FOR i:=1 TO 5 DO
	m_spring2Param[i]:=g_spring2Param[i];
	m_spring3Param[i]:=g_spring3Param[i];
	m_spring5Param[i]:=g_spring5Param[i];
END_FOR
m_spring3Param[6]:=g_spring3Param[6];
END_METHOD

METHOD PUBLIC run : BOOL
VAR_IN_OUT CONSTANT
	// active joint position
	i_jntPos :vec7d;
END_VAR
VAR_IN_OUT
	r_gravity :Vec7d;
END_VAR
VAR

	// position of all the active joint
	m_leftJntPos:ARRAY[1..7] OF LREAL;
	m_rightJntPos:ARRAY[1..7] OF LREAL;
	
	// gravity regression matrix
	regMat:ARRAY[1..5,1..16] OF LREAL;
	
	i,j:INT;
END_VAR
getRegMat(m_armIdx,i_jntPos,regMat);

FOR i:=2 TO 6 DO
	r_gravity[i]:=0;
	FOR j:=1 TO 16 DO
		r_gravity[i]:=r_gravity[i]+regMat[i-1,j]*m_gravityParam[j];
	END_FOR
END_FOR
END_METHOD

(*spring force F = preF+k(L-L0)
% torque trq=F*t=preF*t+k*t*(L-L0)=[t, t*(L-L0)]*[preF,k]'
% this function return [t, t(L-L0)]*)
METHOD PROTECTED spring2RegMat : BOOL
VAR_INPUT
	i_q2:LREAL;
END_VAR

VAR
	// spring paramters
	L0, b1, b2, l1, r0 : LREAL;

	theta,length,t:LREAL;  
	
END_VAR

VAR_OUTPUT
	o_preF:LREAL;
	o_stiff:LREAL;
END_VAR
L0:=m_spring2Param[1]; 
b1:=m_spring2Param[2]; 
b2:=m_spring2Param[3]; 
l1:=m_spring2Param[4]; 
r0:=m_spring2Param[5]; 

L0:=L0+b1+b2;
 
//spring length
theta:=i_q2+90*g_deg2Rad;
length:=SQRT(l1*l1+r0*r0+2*l1*r0*COS(theta));

//force arm
t:=r0*l1*SIN(theta)/Length;

//torque direction is determined by theta(or t)
o_preF:=t;
o_stiff:=t*(length-L0);
END_METHOD

(*spring force F = preF+k(L-L0)
% torque trq=F*t=preF*t+k*t*(L-L0)=[t, t*(L-L0)]*[preF,k]'
% this function return [t, t(L-L0)]*)
METHOD PROTECTED spring3RegMat : BOOL
VAR_INPUT
	i_q3:LREAL;
END_VAR

VAR
	// spring paramters
	L0, b1, b2, l1, r0, d: LREAL;

	alpha, beta,tanBeta, length,t:LREAL;  
	
	spring: INT;
END_VAR

VAR_OUTPUT
	o_preF:LREAL;
	o_stiff:LREAL;
END_VAR
L0:=m_spring3Param[1]; 
b1:=m_spring3Param[2]; 
b2:=m_spring3Param[3]; 
l1:=m_spring3Param[4]; 
r0:=m_spring3Param[5];
d:=m_spring3Param[6];

L0:=L0+b1+b2;
 
// spring length
    alpha:=i_q3+90*g_deg2Rad;
    tanBeta:=(r0*SIN(alpha)+d)/(l1+r0*COS(alpha));
    beta:=ATAN(tanBeta);
    length:=d/SIN(beta)+r0*SIN(alpha)/SIN(beta);
    
// force arm
    t:=(l1-d*cot(beta))*SIN(beta);
    
// torque direction is determined by theta(or t)
    o_preF:=t;
    o_stiff:=t*(length-L0);
END_METHOD

(*spring force F = preF+k(L-L0)
 torque trq=F*t=preF*t+k*t*(L-L0)=[t, t*(L-L0)]*[preF,k]'
 this function return [t, t(L-L0)]
 armIdx, 0 for left arm , 1 for right arm]*)
METHOD PROTECTED spring5RegMat : BOOL
VAR_INPUT
	i_q5:LREAL;
END_VAR

VAR
	// spring paramters
	L0, s1, L1, r0, beta: LREAL;

	theta, length,t:LREAL;  
	
	spring: INT;
	joint: INT;
	armIdx: INT;
	b1: LREAL;
END_VAR

VAR_OUTPUT
	o_preF:LREAL;
	o_stiff:LREAL;
END_VAR
L0:=m_spring5Param[1]; 
s1:=m_spring5Param[2]; 
L1:=m_spring5Param[3]; 
r0:=m_spring5Param[4]; 
beta:=m_spring5Param[5];

L0:=L0+s1;
 
// joint 5 motion angle
IF 1=m_armIdx THEN 
	theta:=i_q5-pi;// left arm
ELSE
	theta:=pi-i_q5; // right arm
END_IF

// spring length and force arm
length:=SQRT(L1*L1+r0*r0+2*L1*r0*COS(theta+beta));
t:=L1*r0*SIN(theta+beta)/length;

// torque direction is determined by t
IF 1=m_armIdx THEN 
	o_preF:=t;
	o_stiff:=t*(length-L0);
else
	o_preF:=-t;
	o_stiff:=-t*(length-L0);
END_IF
END_METHOD

END_FUNCTION_BLOCK

// ---- FBs_RobotDynamics/FB_MasterDynamic.TcPOU
FUNCTION_BLOCK FB_MasterDynamic
VAR_INPUT
END_VAR
VAR_OUTPUT
END_VAR
VAR
	m_armIdx :INT;
	//kinematic constraint
	//  q3 = q8 - q2;            qdot3=qdot8-qdot2;
	//  q9 = q2-q8;              qdot9=qdot2-qdot8;
	//  q4= q4motor+q8-q2-90;    qdot4=qdot4m+qdot8
 	// jacobian with active joints
 	// jaco_DH*qdot_DH = jaco_DH * (A * qdot_active)= jaco * qdot_active
 	// q_DH=[q1,q2,q3,q4,q5,q6,q7,q8,q9];
 	// q_active=[q1,q2,q8,q4m,q5,q6,q7]
	m_jacoA :ARRAY[1..9,1..7] OF LREAL:=
		[   1,  0,  0,  0,  0,  0,  0,
			0,  1,  0,  0,  0,  0,  0,
			0, -1,  1,  0,  0,  0,  0,
			0, -1,  1,  1,  0,  0,  0,
			0,  0,  0,  0,  1,  0,  0,
			0,  0,  0,  0,  0,  1,  0,
			0,  0,  0,  0,  0,  0,  1,
			0,  0,  1,  0,  0,  0,  0,
			0,  1, -1,  0,  0,  0,  0];
	
	// DH parameters
	m_armDH:ARRAY[1..9] OF Vec4d;// last column is joint position
	m_d1, m_a3,m_a4,m_d4,m_a9 :LREAL;
	
	// dynamic parameters
	m_linkMass :ARRAY[1..9] OF LREAL;
	m_linkCOM :ARRAY[1..9] OF Vec3d;
	m_linkInertia :ARRAY[1..9] OF Mat3d;
		
	// frame of each joint
	m_jntFrame :ARRAY[1..9] OF ST_Frame;
	
	// jacobian of mass center
	m_Jp :ARRAY[1..9] OF Mat37;
	m_Jo :ARRAY[1..9] OF Mat37;
	
	// tcp jacobian
	m_jaco : Mat67;
	
	// motor inertia at link size
	m_motorInertia :Vec7d;
	
	// mass matrix in joint space
	m_massMat :Mat7d;
	m_massMatInv:Mat7d;
	
	// mass matrix in cartesian space
	m_lambdaInv :Mat6d;
	m_lambda :Mat6d;
	
	// dynamic nullspace(I-J'*inv(J'))
	m_JtGeneInv :Mat67;
	m_dynaNullspace : Mat7d;
	
END_VAR

PROPERTY PUBLIC cartMassMat : Mat6d
GET
cartMassMat := m_lambda;
END_GET
END_PROPERTY

PROPERTY PUBLIC dynaNullspace : Mat7d
GET
dynaNullspace:=m_dynaNullspace;
END_GET
END_PROPERTY

METHOD init : BOOL
VAR_INPUT
	i_armIdx :INT ;
END_VAR

VAR
	i:INT;
END_VAR
m_armIdx:=i_armIdx;
m_d1:=g_d1;
m_a3:=g_a3;
m_a4:=g_a4;
m_d4:=g_d4;
m_a9:=g_a9;

m_linkMass:=g_linkMass;
FOR i:=1 TO 9 DO
	m_linkCOM[i][1]:=g_linkCOM[i,1];
	m_linkCOM[i][2]:=g_linkCOM[i,2];
	m_linkCOM[i][3]:=g_linkCOM[i,3];
	
	m_armDH[i][1]:=g_masterArmDH[i,1];
	m_armDH[i][2]:=g_masterArmDH[i,2];
	m_armDH[i][3]:=g_masterArmDH[i,3];
	m_armDH[i][4]:=g_masterArmDH[i,4];
	
	m_linkInertia[i][1,1]:=g_linkInertia[i,1];
	m_linkInertia[i][2,2]:=g_linkInertia[i,2];
	m_linkInertia[i][3,3]:=g_linkInertia[i,3];
	m_linkInertia[i][1,2]:=g_linkInertia[i,4];
	m_linkInertia[i][1,3]:=g_linkInertia[i,5];
	m_linkInertia[i][2,3]:=g_linkInertia[i,6];
	m_linkInertia[i][2,1]:=m_linkInertia[i][1,2];
	m_linkInertia[i][3,1]:=m_linkInertia[i][1,3];
	m_linkInertia[i][3,2]:=m_linkInertia[i][2,3];
END_FOR

FOR i:=1 TO 7 DO
	m_motorInertia[i]:=g_motorInertia[i]*g_motorReduction[i]*g_motorReduction[i];
END_FOR
END_METHOD

PROPERTY PUBLIC jntMassMat : Mat7d
GET
jntMassMat := m_massMat;
END_GET
END_PROPERTY

// update dynamic and kinematic data 
METHOD updateDynamic : BOOL
VAR_IN_OUT CONSTANT
	i_jntPos : Vec7d;
END_VAR
VAR
	
	i,j:INT;
	m,n :INT;
	linkMassMat :ARRAY[1..9] OF Mat7d;
	linkInerMat :ARRAY[1..9] OF Mat7d;
	inertia,Rt :Mat3d;
	JotI :ARRAY[1..7,1..3] OF LREAL;
	Jot :ARRAY[1..7,1..3] OF LREAL;
	Jpt :ARRAY[1..7,1..3] OF LREAL;
	
	tmpMat3d :Mat3d;
	tmpMat67: Mat67;
	tmpMat7d : Mat7d;
	jacoT: Mat76;
	
END_VAR
// update kinematic 
updateKinematic(i_jntPos);

// joint space mass matrix
// massMat=m*Jp'*Jp+Jo'*R*I*R'*Jo
FOR i:=1 TO 9 DO
	// iner=R*I*R'
	matMultiply(m_jntFrame[i].m_rot,m_linkInertia[i],tmpMat3d);
	matTranspose(m_jntFrame[i].m_rot, Rt);
	matMultiply(tmpMat3d,Rt,inertia);
	
	// m*Jp'*Jp+Jo'*iner*Jo
	matTranspose(m_Jp[i],Jpt);
	matMultiply(Jpt,m_Jp[i], tmpMat7d);
	matMultiNum(tmpMat7d, m_linkMass[i],linkMassMat[i]);
	
	matTranspose(m_Jo[i],Jot);
	matMultiply(Jot,inertia, JotI);
	matMultiply(JotI,m_Jo[i],linkInerMat[i]);
END_FOR

// total mass mat
m_massMat :=g_zeroMat7d;
FOR i:=1 TO 9 DO
	matSelfAdd(m_massMat,linkMassMat[i]);
	matSelfAdd(m_massMat,linkInerMat[i]);
END_FOR

// add motor inertial 
FOR i:=1 TO 7 DO
	m_massMat[i,i]:=m_massMat[i,i]+m_motorInertia[i];
END_FOR

// mass mat inverse
invMat7(m_massMat,m_massMatInv);

// cartesian mass matrix
matTranspose(m_jaco, jacoT);
matMultiply(m_jaco,m_massMatInv, tmpMat67);
matMultiply(tmpMat67, jacoT, m_lambdaInv);
invMat6(m_lambdaInv, m_lambda);

// dyanmic nullspace
matMultiply(m_lambda, m_jaco, tmpMat67);
matMultiply(tmpMat67, m_massMatInv, m_JtGeneInv);
matMultiply(jacoT,m_JtGeneInv,tmpMat7d);
matSub(g_eye7d, tmpMat7d, m_dynaNullspace);
END_METHOD

// only update kinematic data
METHOD PUBLIC updateKinematic : BOOL
VAR_IN_OUT CONSTANT
	i_jntPos : Vec7d;
END_VAR
VAR
	Jp :ARRAY[1..3, 1..9] OF LREAL:=[27(0)];
	Jo :ARRAY[1..3, 1..9] OF LREAL:=[27(0)];
	jacoDH :Mat67;
	T :ST_Frame;
	i,j:INT;
	Pc,z,p:Vec3d;
	tcpPos :Vec3d;
	m,n :INT;
	
END_VAR
// tranform a joint positon to DH ones
m_armDH[1][4]:=i_jntPos[1];
m_armDH[2][4]:=i_jntPos[2];
m_armDH[3][4]:=i_jntPos[3]-i_jntPos[2];
m_armDH[4][4]:=i_jntPos[4]+i_jntPos[3]-i_jntPos[2]-pi/2;
m_armDH[5][4]:=i_jntPos[5];
m_armDH[6][4]:=i_jntPos[6];
m_armDH[7][4]:=i_jntPos[7];
m_armDH[8][4]:=i_jntPos[3];
m_armDH[9][4]:=i_jntPos[2]-i_jntPos[3];

// compute joint frame
m_jntFrame[1]:=DHTrans(m_armDH[1]);
T:=DHTrans(m_armDH[2]);
m_jntFrame[2]:=transform(m_jntFrame[1],T);
T:=DHTrans(m_armDH[3]);
m_jntFrame[3]:=transform(m_jntFrame[2],T);
T:=DHTrans(m_armDH[4]);
m_jntFrame[4]:=transform(m_jntFrame[3],T);
T:=DHTrans(m_armDH[5]);
m_jntFrame[5]:=transform(m_jntFrame[4],T);
T:=DHTrans(m_armDH[6]);
m_jntFrame[6]:=transform(m_jntFrame[5],T);
T:=DHTrans(m_armDH[7]);
m_jntFrame[7]:=transform(m_jntFrame[6],T);
T:=DHTrans(m_armDH[8]);
m_jntFrame[8]:=transform(m_jntFrame[1],T);
T:=DHTrans(m_armDH[9]);
m_jntFrame[9]:=transform(m_jntFrame[8],T);

// tcp jacobian
tcpPos:=m_jntFrame[7].m_pos;
FOR i:=1 TO 7 DO
	T:=m_jntFrame[i];
	z[1]:=T.m_rot[1,3];
	z[2]:=T.m_rot[2,3];
	z[3]:=T.m_rot[3,3];
	p:=subVec3(tcpPos,T.m_pos);
	p:=cross(z,p);
	jacoDH[1,i]:=p[1];
	jacoDH[2,i]:=p[2];
	jacoDH[3,i]:=p[3];
	jacoDH[4,i]:=z[1];
	jacoDH[5,i]:=z[2];
	jacoDH[6,i]:=z[3];
END_FOR
// multiply m_jacoA
FOR m:=1 TO 6 DO 
	FOR n:=1 TO 7 DO
		IF 2=n THEN
			m_Jaco[m,n]:=jacoDH[m,2]-jacoDH[m,3]-jacoDH[m,4];
		ELSIF 3 =n THEN
			m_Jaco[m,n]:=jacoDH[m,3]+jacoDH[m,4];
		ELSE
			m_Jaco[m,n]:=jacoDH[m,n];
		END_IF
	END_FOR
END_FOR


// jacobian of mass center
FOR i:=1 TO 9 DO 
    T:=m_jntFrame[i];
	// mass center world position
    Pc:=mat3Vec3(T.m_rot,m_linkCOM[i]);
	Pc:=addVec3(Pc,T.m_pos);
    FOR j:=1 TO i DO
        IF (i>7 AND j>1 AND j<8) THEN
			Jp[1,j]:=0;
			Jp[2,j]:=0;
			Jp[3,j]:=0;
			Jo[1,j]:=0;
			Jo[2,j]:=0;
			Jo[3,j]:=0;
            CONTINUE;
        END_IF
        T:=m_jntFrame[j];
		z[1]:=T.m_rot[1,3];
		z[2]:=T.m_rot[2,3];
		z[3]:=T.m_rot[3,3];
        p:=subVec3(Pc,T.m_pos);
		p:=cross(z,p);
		Jp[1,j]:=p[1];
		Jp[2,j]:=p[2];
		Jp[3,j]:=p[3];
        Jo[1,j]:=z[1];
		Jo[2,j]:=z[2];
		Jo[3,j]:=z[3];
    END_FOR
	// multiply m_jacoA
	FOR m:=1 TO 3 DO 
		FOR n:=1 TO 7 DO
			IF 2=n THEN
				m_Jp[i][m,n]:=Jp[m,2]-Jp[m,3]-Jp[m,4]+Jp[m,9];
				m_Jo[i][m,n]:=Jo[m,2]-Jo[m,3]-Jo[m,4]+Jo[m,9];
			ELSIF 3 =n THEN
				m_Jp[i][m,n]:=Jp[m,3]+Jp[m,4]+Jp[m,8]-Jp[m,9];
				m_Jo[i][m,n]:=Jo[m,3]+Jo[m,4]+Jo[m,8]-Jo[m,9];
			ELSE
				m_Jp[i][m,n]:=Jp[m,n];
				m_Jo[i][m,n]:=Jo[m,n];
			END_IF
		END_FOR
	END_FOR
END_FOR
END_METHOD

END_FUNCTION_BLOCK

// ---- MatrixLib/matMultiply.TcPOU
// matC = matA * matB
FUNCTION matMultiply : BOOL
VAR_IN_OUT CONSTANT
	matA :ARRAY[*,*] OF LREAL;//m*p
	matB :ARRAY[*,*] OF LREAL;//p*n
END_VAR

VAR_IN_OUT 
	matC :ARRAY[*,*] OF LREAL;//m*n
END_VAR

VAR
	i,j, k :DINT;
	m,n,p :DINT;
	tmp:LREAL;
 
END_VAR

m:=UPPER_BOUND(matA,1);
p:=UPPER_BOUND(matA,2);
n:=UPPER_BOUND(matB,2);

FOR i:=1 TO m DO
	FOR j:=1 TO n DO
		matC[i,j]:=0.0;
	END_FOR
END_FOR

FOR i:=1 TO m DO
	FOR k:=1 TO p DO
		tmp:=matA[i,k];
		FOR j:=1 TO n DO 
		matC[i,j]:=matC[i,j]+tmp*matB[k,j];
		END_FOR
	END_FOR
END_FOR

END_FUNCTION

// ---- MatrixLib/matTranspose.TcPOU
// B =A'
FUNCTION matTranspose : BOOL
VAR_IN_OUT CONSTANT
	matA :ARRAY[*,*] OF LREAL;
END_VAR

VAR_IN_OUT 
	matB :ARRAY[*,*] OF LREAL;
END_VAR

VAR
	i,j:DINT;
	m,n :DINT;
 
END_VAR

m:=UPPER_BOUND(matB,1);
n:= UPPER_BOUND(matB,2);
FOR i:=1 TO m DO
	FOR j:=1 TO n DO
		matB[i,j]:=matA[j,i];
	END_FOR
END_FOR

END_FUNCTION

// ---- MatrixLib/matMultiNum.TcPOU
// matB=num*MatA
FUNCTION matMultiNum : BOOL
VAR_IN_OUT CONSTANT
	matA :ARRAY[*,*] OF LREAL;
	num : LREAL;
END_VAR

VAR_IN_OUT 
	matB :ARRAY[*,*] OF LREAL;
END_VAR

VAR
	m,n :DINT;
	i,j, k :DINT;
 
END_VAR

m:=UPPER_BOUND(matB,1);
n:= UPPER_BOUND(matB,2);
FOR i:=1 TO m DO
	FOR j:=1 TO n DO
		matB[i,j]:=num*matA[i,j];
	END_FOR
END_FOR

END_FUNCTION

// ---- MatrixLib/invMat7.TcPOU
FUNCTION invMat7 : bool
VAR_IN_OUT CONSTANT
	mat :Mat7d;
END_VAR

VAR_IN_OUT
	invMat :Mat7d;
END_VAR
VAR
	dim : INT :=7;
	i,j,k,h:INT;
	m,n :INT;
	cofactorMat : Mat6d;
	adjointMat :Mat7d;
	matDet :LREAL;
END_VAR

matDet :=Det7(mat);
IF matDet=0 THEN
	invMat7:=FALSE;
	RETURN;
END_IF

FOR i :=1 TO dim DO
	FOR j:=1 TO dim DO
		// get cofactor mat
		m:=1;
		n:=1;
		FOR k:=1 TO dim DO
			FOR h:=1 TO dim DO
				IF k<>i AND h <> j THEN
					cofactorMat[m,n]:=mat[k,h];
					n:=n+1;
					IF n>=dim THEN
						m:=m+1;
						n:=1;
					END_IF
				END_IF
			END_FOR
		END_FOR
		
		adjointMat[i,j]:=EXPT(-1,i+j)*Det6(cofactorMat);
	END_FOR
END_FOR

FOR i :=1 TO dim DO
	FOR j:=1 TO dim DO
		invMat[i,j]:=adjointMat[j,i]/matDet;
	END_FOR
END_FOR
invMat7:=true;

END_FUNCTION

// ---- MatrixLib/Det7.TcPOU
FUNCTION Det7 : LREAL
VAR_IN_OUT CONSTANT
	mat: Mat7d;
END_VAR
VAR
	dim : INT :=7;
	i,j,k:INT;
	m,n :INT;
	cofactorMat : Mat6d;
END_VAR

Det7:=0;
FOR i :=1 TO dim DO
	// get cofactor mat
	m:=1;
	n:=1;
	FOR j:=1 TO dim DO
		FOR k:=1 TO dim DO
			IF j<>1 AND k <> i THEN
				cofactorMat[m,n]:=mat[j,k];
				n:=n+1;
				IF n>=dim THEN
					m:=m+1;
					n:=1;
				END_IF
			END_IF
		END_FOR
	END_FOR
	
	Det7:=Det7+ mat[1,i]*EXPT(-1,1+i)*Det6(cofactorMat);
END_FOR

END_FUNCTION

// ---- MatrixLib/Det6.TcPOU
FUNCTION Det6 : LREAL
VAR_IN_OUT CONSTANT
	mat: Mat6d;
END_VAR
VAR
	a11,a12,a13,a14,a15,a16:LREAL;
	a21,a22,a23,a24,a25,a26:LREAL;
	a31,a32,a33,a34,a35,a36:LREAL;
	a41,a42,a43,a44,a45,a46:LREAL;
	a51,a52,a53,a54,a55,a56:LREAL;
	a61,a62,a63,a64,a65,a66:LREAL;
END_VAR


a11:=mat[1,1];
a12:=mat[1,2];
a13:=mat[1,3];
a14:=mat[1,4];
a15:=mat[1,5];
a16:=mat[1,6];

a21:=mat[2,1];
a22:=mat[2,2];
a23:=mat[2,3];
a24:=mat[2,4];
a25:=mat[2,5];
a26:=mat[2,6];

a31:=mat[3,1];
a32:=mat[3,2];
a33:=mat[3,3];
a34:=mat[3,4];
a35:=mat[3,5];
a36:=mat[3,6];

a41:=mat[4,1];
a42:=mat[4,2];
a43:=mat[4,3];
a44:=mat[4,4];
a45:=mat[4,5];
a46:=mat[4,6];

a51:=mat[5,1];
a52:=mat[5,2];
a53:=mat[5,3];
a54:=mat[5,4];
a55:=mat[5,5];
a56:=mat[5,6];

a61:=mat[6,1];
a62:=mat[6,2];
a63:=mat[6,3];
a64:=mat[6,4];
a65:=mat[6,5];
a66:=mat[6,6];

//Det6:=a11*a22*a33*a44*a55*a66 - a11*a22*a33*a44*a56*a65 - a11*a22*a33*a45*a54*a66 + a11*a22*a33*a45*a56*a64 + a11*a22*a33*a46*a54*a65 - a11*a22*a33*a46*a55*a64 - a11*a22*a34*a43*a55*a66 + a11*a22*a34*a43*a56*a65 + a11*a22*a34*a45*a53*a66 - a11*a22*a34*a45*a56*a63 - a11*a22*a34*a46*a53*a65 + a11*a22*a34*a46*a55*a63 + a11*a22*a35*a43*a54*a66 - a11*a22*a35*a43*a56*a64 - a11*a22*a35*a44*a53*a66 + a11*a22*a35*a44*a56*a63 + a11*a22*a35*a46*a53*a64 - a11*a22*a35*a46*a54*a63 - a11*a22*a36*a43*a54*a65 + a11*a22*a36*a43*a55*a64 + a11*a22*a36*a44*a53*a65 - a11*a22*a36*a44*a55*a63 - a11*a22*a36*a45*a53*a64 + a11*a22*a36*a45*a54*a63 - a11*a23*a32*a44*a55*a66 + a11*a23*a32*a44*a56*a65 + a11*a23*a32*a45*a54*a66 - a11*a23*a32*a45*a56*a64 - a11*a23*a32*a46*a54*a65 + a11*a23*a32*a46*a55*a64 + a11*a23*a34*a42*a55*a66 - a11*a23*a34*a42*a56*a65 - a11*a23*a34*a45*a52*a66 + a11*a23*a34*a45*a56*a62 + a11*a23*a34*a46*a52*a65 - a11*a23*a34*a46*a55*a62 - a11*a23*a35*a42*a54*a66 + a11*a23*a35*a42*a56*a64 + a11*a23*a35*a44*a52*a66 - a11*a23*a35*a44*a56*a62 - a11*a23*a35*a46*a52*a64 + a11*a23*a35*a46*a54*a62 + a11*a23*a36*a42*a54*a65 - a11*a23*a36*a42*a55*a64 - a11*a23*a36*a44*a52*a65 + a11*a23*a36*a44*a55*a62 + a11*a23*a36*a45*a52*a64 - a11*a23*a36*a45*a54*a62 + a11*a24*a32*a43*a55*a66 - a11*a24*a32*a43*a56*a65 - a11*a24*a32*a45*a53*a66 + a11*a24*a32*a45*a56*a63 + a11*a24*a32*a46*a53*a65 - a11*a24*a32*a46*a55*a63 - a11*a24*a33*a42*a55*a66 + a11*a24*a33*a42*a56*a65 + a11*a24*a33*a45*a52*a66 - a11*a24*a33*a45*a56*a62 - a11*a24*a33*a46*a52*a65 + a11*a24*a33*a46*a55*a62 + a11*a24*a35*a42*a53*a66 - a11*a24*a35*a42*a56*a63 - a11*a24*a35*a43*a52*a66 + a11*a24*a35*a43*a56*a62 + a11*a24*a35*a46*a52*a63 - a11*a24*a35*a46*a53*a62 - a11*a24*a36*a42*a53*a65 + a11*a24*a36*a42*a55*a63 + a11*a24*a36*a43*a52*a65 - a11*a24*a36*a43*a55*a62 - a11*a24*a36*a45*a52*a63 + a11*a24*a36*a45*a53*a62 - a11*a25*a32*a43*a54*a66 + a11*a25*a32*a43*a56*a64 + a11*a25*a32*a44*a53*a66 - a11*a25*a32*a44*a56*a63 - a11*a25*a32*a46*a53*a64 + a11*a25*a32*a46*a54*a63 + a11*a25*a33*a42*a54*a66 - a11*a25*a33*a42*a56*a64 - a11*a25*a33*a44*a52*a66 + a11*a25*a33*a44*a56*a62 + a11*a25*a33*a46*a52*a64 - a11*a25*a33*a46*a54*a62 - a11*a25*a34*a42*a53*a66 + a11*a25*a34*a42*a56*a63 + a11*a25*a34*a43*a52*a66 - a11*a25*a34*a43*a56*a62 - a11*a25*a34*a46*a52*a63 + a11*a25*a34*a46*a53*a62 + a11*a25*a36*a42*a53*a64 - a11*a25*a36*a42*a54*a63 - a11*a25*a36*a43*a52*a64 + a11*a25*a36*a43*a54*a62 + a11*a25*a36*a44*a52*a63 - a11*a25*a36*a44*a53*a62 + a11*a26*a32*a43*a54*a65 - a11*a26*a32*a43*a55*a64 - a11*a26*a32*a44*a53*a65 + a11*a26*a32*a44*a55*a63 + a11*a26*a32*a45*a53*a64 - a11*a26*a32*a45*a54*a63 - a11*a26*a33*a42*a54*a65 + a11*a26*a33*a42*a55*a64 + a11*a26*a33*a44*a52*a65 - a11*a26*a33*a44*a55*a62 - a11*a26*a33*a45*a52*a64 + a11*a26*a33*a45*a54*a62 + a11*a26*a34*a42*a53*a65 - a11*a26*a34*a42*a55*a63 - a11*a26*a34*a43*a52*a65 + a11*a26*a34*a43*a55*a62 + a11*a26*a34*a45*a52*a63 - a11*a26*a34*a45*a53*a62 - a11*a26*a35*a42*a53*a64 + a11*a26*a35*a42*a54*a63 + a11*a26*a35*a43*a52*a64 - a11*a26*a35*a43*a54*a62 - a11*a26*a35*a44*a52*a63 + a11*a26*a35*a44*a53*a62 - a12*a21*a33*a44*a55*a66 + a12*a21*a33*a44*a56*a65 + a12*a21*a33*a45*a54*a66 - a12*a21*a33*a45*a56*a64 - a12*a21*a33*a46*a54*a65 + a12*a21*a33*a46*a55*a64 + a12*a21*a34*a43*a55*a66 - a12*a21*a34*a43*a56*a65 - a12*a21*a34*a45*a53*a66 + a12*a21*a34*a45*a56*a63 + a12*a21*a34*a46*a53*a65 - a12*a21*a34*a46*a55*a63 - a12*a21*a35*a43*a54*a66 + a12*a21*a35*a43*a56*a64 + a12*a21*a35*a44*a53*a66 - a12*a21*a35*a44*a56*a63 - a12*a21*a35*a46*a53*a64 + a12*a21*a35*a46*a54*a63 + a12*a21*a36*a43*a54*a65 - a12*a21*a36*a43*a55*a64 - a12*a21*a36*a44*a53*a65 + a12*a21*a36*a44*a55*a63 + a12*a21*a36*a45*a53*a64 - a12*a21*a36*a45*a54*a63 + a12*a23*a31*a44*a55*a66 - a12*a23*a31*a44*a56*a65 - a12*a23*a31*a45*a54*a66 + a12*a23*a31*a45*a56*a64 + a12*a23*a31*a46*a54*a65 - a12*a23*a31*a46*a55*a64 - a12*a23*a34*a41*a55*a66 + a12*a23*a34*a41*a56*a65 + a12*a23*a34*a45*a51*a66 - a12*a23*a34*a45*a56*a61 - a12*a23*a34*a46*a51*a65 + a12*a23*a34*a46*a55*a61 + a12*a23*a35*a41*a54*a66 - a12*a23*a35*a41*a56*a64 - a12*a23*a35*a44*a51*a66 + a12*a23*a35*a44*a56*a61 + a12*a23*a35*a46*a51*a64 - a12*a23*a35*a46*a54*a61 - a12*a23*a36*a41*a54*a65 + a12*a23*a36*a41*a55*a64 + a12*a23*a36*a44*a51*a65 - a12*a23*a36*a44*a55*a61 - a12*a23*a36*a45*a51*a64 + a12*a23*a36*a45*a54*a61 - a12*a24*a31*a43*a55*a66 + a12*a24*a31*a43*a56*a65 + a12*a24*a31*a45*a53*a66 - a12*a24*a31*a45*a56*a63 - a12*a24*a31*a46*a53*a65 + a12*a24*a31*a46*a55*a63 + a12*a24*a33*a41*a55*a66 - a12*a24*a33*a41*a56*a65 - a12*a24*a33*a45*a51*a66 + a12*a24*a33*a45*a56*a61 + a12*a24*a33*a46*a51*a65 - a12*a24*a33*a46*a55*a61 - a12*a24*a35*a41*a53*a66 + a12*a24*a35*a41*a56*a63 + a12*a24*a35*a43*a51*a66 - a12*a24*a35*a43*a56*a61 - a12*a24*a35*a46*a51*a63 + a12*a24*a35*a46*a53*a61 + a12*a24*a36*a41*a53*a65 - a12*a24*a36*a41*a55*a63 - a12*a24*a36*a43*a51*a65 + a12*a24*a36*a43*a55*a61 + a12*a24*a36*a45*a51*a63 - a12*a24*a36*a45*a53*a61 + a12*a25*a31*a43*a54*a66 - a12*a25*a31*a43*a56*a64 - a12*a25*a31*a44*a53*a66 + a12*a25*a31*a44*a56*a63 + a12*a25*a31*a46*a53*a64 - a12*a25*a31*a46*a54*a63 - a12*a25*a33*a41*a54*a66 + a12*a25*a33*a41*a56*a64 + a12*a25*a33*a44*a51*a66 - a12*a25*a33*a44*a56*a61 - a12*a25*a33*a46*a51*a64 + a12*a25*a33*a46*a54*a61 + a12*a25*a34*a41*a53*a66 - a12*a25*a34*a41*a56*a63 - a12*a25*a34*a43*a51*a66 + a12*a25*a34*a43*a56*a61 + a12*a25*a34*a46*a51*a63 - a12*a25*a34*a46*a53*a61 - a12*a25*a36*a41*a53*a64 + a12*a25*a36*a41*a54*a63 + a12*a25*a36*a43*a51*a64 - a12*a25*a36*a43*a54*a61 - a12*a25*a36*a44*a51*a63 + a12*a25*a36*a44*a53*a61 - a12*a26*a31*a43*a54*a65 + a12*a26*a31*a43*a55*a64 + a12*a26*a31*a44*a53*a65 - a12*a26*a31*a44*a55*a63 - a12*a26*a31*a45*a53*a64 + a12*a26*a31*a45*a54*a63 + a12*a26*a33*a41*a54*a65 - a12*a26*a33*a41*a55*a64 - a12*a26*a33*a44*a51*a65 + a12*a26*a33*a44*a55*a61 + a12*a26*a33*a45*a51*a64 - a12*a26*a33*a45*a54*a61 - a12*a26*a34*a41*a53*a65 + a12*a26*a34*a41*a55*a63 + a12*a26*a34*a43*a51*a65 - a12*a26*a34*a43*a55*a61 - a12*a26*a34*a45*a51*a63 + a12*a26*a34*a45*a53*a61 + a12*a26*a35*a41*a53*a64 - a12*a26*a35*a41*a54*a63 - a12*a26*a35*a43*a51*a64 + a12*a26*a35*a43*a54*a61 + a12*a26*a35*a44*a51*a63 - a12*a26*a35*a44*a53*a61 + a13*a21*a32*a44*a55*a66 - a13*a21*a32*a44*a56*a65 - a13*a21*a32*a45*a54*a66 + a13*a21*a32*a45*a56*a64 + a13*a21*a32*a46*a54*a65 - a13*a21*a32*a46*a55*a64 - a13*a21*a34*a42*a55*a66 + a13*a21*a34*a42*a56*a65 + a13*a21*a34*a45*a52*a66 - a13*a21*a34*a45*a56*a62 - a13*a21*a34*a46*a52*a65 + a13*a21*a34*a46*a55*a62 + a13*a21*a35*a42*a54*a66 - a13*a21*a35*a42*a56*a64 - a13*a21*a35*a44*a52*a66 + a13*a21*a35*a44*a56*a62 + a13*a21*a35*a46*a52*a64 - a13*a21*a35*a46*a54*a62 - a13*a21*a36*a42*a54*a65 + a13*a21*a36*a42*a55*a64 + a13*a21*a36*a44*a52*a65 - a13*a21*a36*a44*a55*a62 - a13*a21*a36*a45*a52*a64 + a13*a21*a36*a45*a54*a62 - a13*a22*a31*a44*a55*a66 + a13*a22*a31*a44*a56*a65 + a13*a22*a31*a45*a54*a66 - a13*a22*a31*a45*a56*a64 - a13*a22*a31*a46*a54*a65 + a13*a22*a31*a46*a55*a64 + a13*a22*a34*a41*a55*a66 - a13*a22*a34*a41*a56*a65 - a13*a22*a34*a45*a51*a66 + a13*a22*a34*a45*a56*a61 + a13*a22*a34*a46*a51*a65 - a13*a22*a34*a46*a55*a61 - a13*a22*a35*a41*a54*a66 + a13*a22*a35*a41*a56*a64 + a13*a22*a35*a44*a51*a66 - a13*a22*a35*a44*a56*a61 - a13*a22*a35*a46*a51*a64 + a13*a22*a35*a46*a54*a61 + a13*a22*a36*a41*a54*a65 - a13*a22*a36*a41*a55*a64 - a13*a22*a36*a44*a51*a65 + a13*a22*a36*a44*a55*a61 + a13*a22*a36*a45*a51*a64 - a13*a22*a36*a45*a54*a61 + a13*a24*a31*a42*a55*a66 - a13*a24*a31*a42*a56*a65 - a13*a24*a31*a45*a52*a66 + a13*a24*a31*a45*a56*a62 + a13*a24*a31*a46*a52*a65 - a13*a24*a31*a46*a55*a62 - a13*a24*a32*a41*a55*a66 + a13*a24*a32*a41*a56*a65 + a13*a24*a32*a45*a51*a66 - a13*a24*a32*a45*a56*a61 - a13*a24*a32*a46*a51*a65 + a13*a24*a32*a46*a55*a61 + a13*a24*a35*a41*a52*a66 - a13*a24*a35*a41*a56*a62 - a13*a24*a35*a42*a51*a66 + a13*a24*a35*a42*a56*a61 + a13*a24*a35*a46*a51*a62 - a13*a24*a35*a46*a52*a61 - a13*a24*a36*a41*a52*a65 + a13*a24*a36*a41*a55*a62 + a13*a24*a36*a42*a51*a65 - a13*a24*a36*a42*a55*a61 - a13*a24*a36*a45*a51*a62 + a13*a24*a36*a45*a52*a61 - a13*a25*a31*a42*a54*a66 + a13*a25*a31*a42*a56*a64 + a13*a25*a31*a44*a52*a66 - a13*a25*a31*a44*a56*a62 - a13*a25*a31*a46*a52*a64 + a13*a25*a31*a46*a54*a62 + a13*a25*a32*a41*a54*a66 - a13*a25*a32*a41*a56*a64 - a13*a25*a32*a44*a51*a66 + a13*a25*a32*a44*a56*a61 + a13*a25*a32*a46*a51*a64 - a13*a25*a32*a46*a54*a61 - a13*a25*a34*a41*a52*a66 + a13*a25*a34*a41*a56*a62 + a13*a25*a34*a42*a51*a66 - a13*a25*a34*a42*a56*a61 - a13*a25*a34*a46*a51*a62 + a13*a25*a34*a46*a52*a61 + a13*a25*a36*a41*a52*a64 - a13*a25*a36*a41*a54*a62 - a13*a25*a36*a42*a51*a64 + a13*a25*a36*a42*a54*a61 + a13*a25*a36*a44*a51*a62 - a13*a25*a36*a44*a52*a61 + a13*a26*a31*a42*a54*a65 - a13*a26*a31*a42*a55*a64 - a13*a26*a31*a44*a52*a65 + a13*a26*a31*a44*a55*a62 + a13*a26*a31*a45*a52*a64 - a13*a26*a31*a45*a54*a62 - a13*a26*a32*a41*a54*a65 + a13*a26*a32*a41*a55*a64 + a13*a26*a32*a44*a51*a65 - a13*a26*a32*a44*a55*a61 - a13*a26*a32*a45*a51*a64 + a13*a26*a32*a45*a54*a61 + a13*a26*a34*a41*a52*a65 - a13*a26*a34*a41*a55*a62 - a13*a26*a34*a42*a51*a65 + a13*a26*a34*a42*a55*a61 + a13*a26*a34*a45*a51*a62 - a13*a26*a34*a45*a52*a61 - a13*a26*a35*a41*a52*a64 + a13*a26*a35*a41*a54*a62 + a13*a26*a35*a42*a51*a64 - a13*a26*a35*a42*a54*a61 - a13*a26*a35*a44*a51*a62 + a13*a26*a35*a44*a52*a61 - a14*a21*a32*a43*a55*a66 + a14*a21*a32*a43*a56*a65 + a14*a21*a32*a45*a53*a66 - a14*a21*a32*a45*a56*a63 - a14*a21*a32*a46*a53*a65 + a14*a21*a32*a46*a55*a63 + a14*a21*a33*a42*a55*a66 - a14*a21*a33*a42*a56*a65 - a14*a21*a33*a45*a52*a66 + a14*a21*a33*a45*a56*a62 + a14*a21*a33*a46*a52*a65 - a14*a21*a33*a46*a55*a62 - a14*a21*a35*a42*a53*a66 + a14*a21*a35*a42*a56*a63 + a14*a21*a35*a43*a52*a66 - a14*a21*a35*a43*a56*a62 - a14*a21*a35*a46*a52*a63 + a14*a21*a35*a46*a53*a62 + a14*a21*a36*a42*a53*a65 - a14*a21*a36*a42*a55*a63 - a14*a21*a36*a43*a52*a65 + a14*a21*a36*a43*a55*a62 + a14*a21*a36*a45*a52*a63 - a14*a21*a36*a45*a53*a62 + a14*a22*a31*a43*a55*a66 - a14*a22*a31*a43*a56*a65 - a14*a22*a31*a45*a53*a66 + a14*a22*a31*a45*a56*a63 + a14*a22*a31*a46*a53*a65 - a14*a22*a31*a46*a55*a63 - a14*a22*a33*a41*a55*a66 + a14*a22*a33*a41*a56*a65 + a14*a22*a33*a45*a51*a66 - a14*a22*a33*a45*a56*a61 - a14*a22*a33*a46*a51*a65 + a14*a22*a33*a46*a55*a61 + a14*a22*a35*a41*a53*a66 - a14*a22*a35*a41*a56*a63 - a14*a22*a35*a43*a51*a66 + a14*a22*a35*a43*a56*a61 + a14*a22*a35*a46*a51*a63 - a14*a22*a35*a46*a53*a61 - a14*a22*a36*a41*a53*a65 + a14*a22*a36*a41*a55*a63 + a14*a22*a36*a43*a51*a65 - a14*a22*a36*a43*a55*a61 - a14*a22*a36*a45*a51*a63 + a14*a22*a36*a45*a53*a61 - a14*a23*a31*a42*a55*a66 + a14*a23*a31*a42*a56*a65 + a14*a23*a31*a45*a52*a66 - a14*a23*a31*a45*a56*a62 - a14*a23*a31*a46*a52*a65 + a14*a23*a31*a46*a55*a62 + a14*a23*a32*a41*a55*a66 - a14*a23*a32*a41*a56*a65 - a14*a23*a32*a45*a51*a66 + a14*a23*a32*a45*a56*a61 + a14*a23*a32*a46*a51*a65 - a14*a23*a32*a46*a55*a61 - a14*a23*a35*a41*a52*a66 + a14*a23*a35*a41*a56*a62 + a14*a23*a35*a42*a51*a66 - a14*a23*a35*a42*a56*a61 - a14*a23*a35*a46*a51*a62 + a14*a23*a35*a46*a52*a61 + a14*a23*a36*a41*a52*a65 - a14*a23*a36*a41*a55*a62 - a14*a23*a36*a42*a51*a65 + a14*a23*a36*a42*a55*a61 + a14*a23*a36*a45*a51*a62 - a14*a23*a36*a45*a52*a61 + a14*a25*a31*a42*a53*a66 - a14*a25*a31*a42*a56*a63 - a14*a25*a31*a43*a52*a66 + a14*a25*a31*a43*a56*a62 + a14*a25*a31*a46*a52*a63 - a14*a25*a31*a46*a53*a62 - a14*a25*a32*a41*a53*a66 + a14*a25*a32*a41*a56*a63 + a14*a25*a32*a43*a51*a66 - a14*a25*a32*a43*a56*a61 - a14*a25*a32*a46*a51*a63 + a14*a25*a32*a46*a53*a61 + a14*a25*a33*a41*a52*a66 - a14*a25*a33*a41*a56*a62 - a14*a25*a33*a42*a51*a66 + a14*a25*a33*a42*a56*a61 + a14*a25*a33*a46*a51*a62 - a14*a25*a33*a46*a52*a61 - a14*a25*a36*a41*a52*a63 + a14*a25*a36*a41*a53*a62 + a14*a25*a36*a42*a51*a63 - a14*a25*a36*a42*a53*a61 - a14*a25*a36*a43*a51*a62 + a14*a25*a36*a43*a52*a61 - a14*a26*a31*a42*a53*a65 + a14*a26*a31*a42*a55*a63 + a14*a26*a31*a43*a52*a65 - a14*a26*a31*a43*a55*a62 - a14*a26*a31*a45*a52*a63 + a14*a26*a31*a45*a53*a62 + a14*a26*a32*a41*a53*a65 - a14*a26*a32*a41*a55*a63 - a14*a26*a32*a43*a51*a65 + a14*a26*a32*a43*a55*a61 + a14*a26*a32*a45*a51*a63 - a14*a26*a32*a45*a53*a61 - a14*a26*a33*a41*a52*a65 + a14*a26*a33*a41*a55*a62 + a14*a26*a33*a42*a51*a65 - a14*a26*a33*a42*a55*a61 - a14*a26*a33*a45*a51*a62 + a14*a26*a33*a45*a52*a61 + a14*a26*a35*a41*a52*a63 - a14*a26*a35*a41*a53*a62 - a14*a26*a35*a42*a51*a63 + a14*a26*a35*a42*a53*a61 + a14*a26*a35*a43*a51*a62 - a14*a26*a35*a43*a52*a61 + a15*a21*a32*a43*a54*a66 - a15*a21*a32*a43*a56*a64 - a15*a21*a32*a44*a53*a66 + a15*a21*a32*a44*a56*a63 + a15*a21*a32*a46*a53*a64 - a15*a21*a32*a46*a54*a63 - a15*a21*a33*a42*a54*a66 + a15*a21*a33*a42*a56*a64 + a15*a21*a33*a44*a52*a66 - a15*a21*a33*a44*a56*a62 - a15*a21*a33*a46*a52*a64 + a15*a21*a33*a46*a54*a62 + a15*a21*a34*a42*a53*a66 - a15*a21*a34*a42*a56*a63 - a15*a21*a34*a43*a52*a66 + a15*a21*a34*a43*a56*a62 + a15*a21*a34*a46*a52*a63 - a15*a21*a34*a46*a53*a62 - a15*a21*a36*a42*a53*a64 + a15*a21*a36*a42*a54*a63 + a15*a21*a36*a43*a52*a64 - a15*a21*a36*a43*a54*a62 - a15*a21*a36*a44*a52*a63 + a15*a21*a36*a44*a53*a62 - a15*a22*a31*a43*a54*a66 + a15*a22*a31*a43*a56*a64 + a15*a22*a31*a44*a53*a66 - a15*a22*a31*a44*a56*a63 - a15*a22*a31*a46*a53*a64 + a15*a22*a31*a46*a54*a63 + a15*a22*a33*a41*a54*a66 - a15*a22*a33*a41*a56*a64 - a15*a22*a33*a44*a51*a66 + a15*a22*a33*a44*a56*a61 + a15*a22*a33*a46*a51*a64 - a15*a22*a33*a46*a54*a61 - a15*a22*a34*a41*a53*a66 + a15*a22*a34*a41*a56*a63 + a15*a22*a34*a43*a51*a66 - a15*a22*a34*a43*a56*a61 - a15*a22*a34*a46*a51*a63 + a15*a22*a34*a46*a53*a61 + a15*a22*a36*a41*a53*a64 - a15*a22*a36*a41*a54*a63 - a15*a22*a36*a43*a51*a64 + a15*a22*a36*a43*a54*a61 + a15*a22*a36*a44*a51*a63 - a15*a22*a36*a44*a53*a61 + a15*a23*a31*a42*a54*a66 - a15*a23*a31*a42*a56*a64 - a15*a23*a31*a44*a52*a66 + a15*a23*a31*a44*a56*a62 + a15*a23*a31*a46*a52*a64 - a15*a23*a31*a46*a54*a62 - a15*a23*a32*a41*a54*a66 + a15*a23*a32*a41*a56*a64 + a15*a23*a32*a44*a51*a66 - a15*a23*a32*a44*a56*a61 - a15*a23*a32*a46*a51*a64 + a15*a23*a32*a46*a54*a61 + a15*a23*a34*a41*a52*a66 - a15*a23*a34*a41*a56*a62 - a15*a23*a34*a42*a51*a66 + a15*a23*a34*a42*a56*a61 + a15*a23*a34*a46*a51*a62 - a15*a23*a34*a46*a52*a61 - a15*a23*a36*a41*a52*a64 + a15*a23*a36*a41*a54*a62 + a15*a23*a36*a42*a51*a64 - a15*a23*a36*a42*a54*a61 - a15*a23*a36*a44*a51*a62 + a15*a23*a36*a44*a52*a61 - a15*a24*a31*a42*a53*a66 + a15*a24*a31*a42*a56*a63 + a15*a24*a31*a43*a52*a66 - a15*a24*a31*a43*a56*a62 - a15*a24*a31*a46*a52*a63 + a15*a24*a31*a46*a53*a62 + a15*a24*a32*a41*a53*a66 - a15*a24*a32*a41*a56*a63 - a15*a24*a32*a43*a51*a66 + a15*a24*a32*a43*a56*a61 + a15*a24*a32*a46*a51*a63 - a15*a24*a32*a46*a53*a61 - a15*a24*a33*a41*a52*a66 + a15*a24*a33*a41*a56*a62 + a15*a24*a33*a42*a51*a66 - a15*a24*a33*a42*a56*a61 - a15*a24*a33*a46*a51*a62 + a15*a24*a33*a46*a52*a61 + a15*a24*a36*a41*a52*a63 - a15*a24*a36*a41*a53*a62 - a15*a24*a36*a42*a51*a63 + a15*a24*a36*a42*a53*a61 + a15*a24*a36*a43*a51*a62 - a15*a24*a36*a43*a52*a61 + a15*a26*a31*a42*a53*a64 - a15*a26*a31*a42*a54*a63 - a15*a26*a31*a43*a52*a64 + a15*a26*a31*a43*a54*a62 + a15*a26*a31*a44*a52*a63 - a15*a26*a31*a44*a53*a62 - a15*a26*a32*a41*a53*a64 + a15*a26*a32*a41*a54*a63 + a15*a26*a32*a43*a51*a64 - a15*a26*a32*a43*a54*a61 - a15*a26*a32*a44*a51*a63 + a15*a26*a32*a44*a53*a61 + a15*a26*a33*a41*a52*a64 - a15*a26*a33*a41*a54*a62 - a15*a26*a33*a42*a51*a64 + a15*a26*a33*a42*a54*a61 + a15*a26*a33*a44*a51*a62 - a15*a26*a33*a44*a52*a61 - a15*a26*a34*a41*a52*a63 + a15*a26*a34*a41*a53*a62 + a15*a26*a34*a42*a51*a63 - a15*a26*a34*a42*a53*a61 - a15*a26*a34*a43*a51*a62 + a15*a26*a34*a43*a52*a61 - a16*a21*a32*a43*a54*a65 + a16*a21*a32*a43*a55*a64 + a16*a21*a32*a44*a53*a65 - a16*a21*a32*a44*a55*a63 - a16*a21*a32*a45*a53*a64 + a16*a21*a32*a45*a54*a63 + a16*a21*a33*a42*a54*a65 - a16*a21*a33*a42*a55*a64 - a16*a21*a33*a44*a52*a65 + a16*a21*a33*a44*a55*a62 + a16*a21*a33*a45*a52*a64 - a16*a21*a33*a45*a54*a62 - a16*a21*a34*a42*a53*a65 + a16*a21*a34*a42*a55*a63 + a16*a21*a34*a43*a52*a65 - a16*a21*a34*a43*a55*a62 - a16*a21*a34*a45*a52*a63 + a16*a21*a34*a45*a53*a62 + a16*a21*a35*a42*a53*a64 - a16*a21*a35*a42*a54*a63 - a16*a21*a35*a43*a52*a64 + a16*a21*a35*a43*a54*a62 + a16*a21*a35*a44*a52*a63 - a16*a21*a35*a44*a53*a62 + a16*a22*a31*a43*a54*a65 - a16*a22*a31*a43*a55*a64 - a16*a22*a31*a44*a53*a65 + a16*a22*a31*a44*a55*a63 + a16*a22*a31*a45*a53*a64 - a16*a22*a31*a45*a54*a63 - a16*a22*a33*a41*a54*a65 + a16*a22*a33*a41*a55*a64 + a16*a22*a33*a44*a51*a65 - a16*a22*a33*a44*a55*a61 - a16*a22*a33*a45*a51*a64 + a16*a22*a33*a45*a54*a61 + a16*a22*a34*a41*a53*a65 - a16*a22*a34*a41*a55*a63 - a16*a22*a34*a43*a51*a65 + a16*a22*a34*a43*a55*a61 + a16*a22*a34*a45*a51*a63 - a16*a22*a34*a45*a53*a61 - a16*a22*a35*a41*a53*a64 + a16*a22*a35*a41*a54*a63 + a16*a22*a35*a43*a51*a64 - a16*a22*a35*a43*a54*a61 - a16*a22*a35*a44*a51*a63 + a16*a22*a35*a44*a53*a61 - a16*a23*a31*a42*a54*a65 + a16*a23*a31*a42*a55*a64 + a16*a23*a31*a44*a52*a65 - a16*a23*a31*a44*a55*a62 - a16*a23*a31*a45*a52*a64 + a16*a23*a31*a45*a54*a62 + a16*a23*a32*a41*a54*a65 - a16*a23*a32*a41*a55*a64 - a16*a23*a32*a44*a51*a65 + a16*a23*a32*a44*a55*a61 + a16*a23*a32*a45*a51*a64 - a16*a23*a32*a45*a54*a61 - a16*a23*a34*a41*a52*a65 + a16*a23*a34*a41*a55*a62 + a16*a23*a34*a42*a51*a65 - a16*a23*a34*a42*a55*a61 - a16*a23*a34*a45*a51*a62 + a16*a23*a34*a45*a52*a61 + a16*a23*a35*a41*a52*a64 - a16*a23*a35*a41*a54*a62 - a16*a23*a35*a42*a51*a64 + a16*a23*a35*a42*a54*a61 + a16*a23*a35*a44*a51*a62 - a16*a23*a35*a44*a52*a61 + a16*a24*a31*a42*a53*a65 - a16*a24*a31*a42*a55*a63 - a16*a24*a31*a43*a52*a65 + a16*a24*a31*a43*a55*a62 + a16*a24*a31*a45*a52*a63 - a16*a24*a31*a45*a53*a62 - a16*a24*a32*a41*a53*a65 + a16*a24*a32*a41*a55*a63 + a16*a24*a32*a43*a51*a65 - a16*a24*a32*a43*a55*a61 - a16*a24*a32*a45*a51*a63 + a16*a24*a32*a45*a53*a61 + a16*a24*a33*a41*a52*a65 - a16*a24*a33*a41*a55*a62 - a16*a24*a33*a42*a51*a65 + a16*a24*a33*a42*a55*a61 + a16*a24*a33*a45*a51*a62 - a16*a24*a33*a45*a52*a61 - a16*a24*a35*a41*a52*a63 + a16*a24*a35*a41*a53*a62 + a16*a24*a35*a42*a51*a63 - a16*a24*a35*a42*a53*a61 - a16*a24*a35*a43*a51*a62 + a16*a24*a35*a43*a52*a61 - a16*a25*a31*a42*a53*a64 + a16*a25*a31*a42*a54*a63 + a16*a25*a31*a43*a52*a64 - a16*a25*a31*a43*a54*a62 - a16*a25*a31*a44*a52*a63 + a16*a25*a31*a44*a53*a62 + a16*a25*a32*a41*a53*a64 - a16*a25*a32*a41*a54*a63 - a16*a25*a32*a43*a51*a64 + a16*a25*a32*a43*a54*a61 + a16*a25*a32*a44*a51*a63 - a16*a25*a32*a44*a53*a61 - a16*a25*a33*a41*a52*a64 + a16*a25*a33*a41*a54*a62 + a16*a25*a33*a42*a51*a64 - a16*a25*a33*a42*a54*a61 - a16*a25*a33*a44*a51*a62 + a16*a25*a33*a44*a52*a61 + a16*a25*a34*a41*a52*a63 - a16*a25*a34*a41*a53*a62 - a16*a25*a34*a42*a51*a63 + a16*a25*a34*a42*a53*a61 + a16*a25*a34*a43*a51*a62 - a16*a25*a34*a43*a52*a61;
Det6:=((a31*a42*a54*a63 - a31*a42*a53*a64 + a31*a43*a52*a64 - a31*a43*a54*a62 - a31*a44*a52*a63 + a31*a44*a53*a62 + a32*a41*a53*a64 - a32*a41*a54*a63 - a32*a43*a51*a64 + a32*a43*a54*a61 + a32*a44*a51*a63 - a32*a44*a53*a61 - a33*a41*a52*a64 + a33*a41*a54*a62 + a33*a42*a51*a64 - a33*a42*a54*a61 - a33*a44*a51*a62 + a33*a44*a52*a61 + a34*a41*a52*a63 - a34*a41*a53*a62 - a34*a42*a51*a63 + a34*a42*a53*a61 + a34*a43*a51*a62 - a34*a43*a52*a61)*a25 + (a31*a42*a53*a65 - a31*a42*a55*a63 - a31*a43*a52*a65 + a31*a43*a55*a62 + a31*a45*a52*a63 - a31*a45*a53*a62 - a32*a41*a53*a65 + a32*a41*a55*a63 + a32*a43*a51*a65 - a32*a43*a55*a61 - a32*a45*a51*a63 + a32*a45*a53*a61 + a33*a41*a52*a65 - a33*a41*a55*a62 - a33*a42*a51*a65 + a33*a42*a55*a61 + a33*a45*a51*a62 - a33*a45*a52*a61 - a35*a41*a52*a63 + a35*a41*a53*a62 + a35*a42*a51*a63 - a35*a42*a53*a61 - a35*a43*a51*a62 + a35*a43*a52*a61)*a24 + (a31*a42*a55*a64 - a31*a42*a54*a65 + a31*a44*a52*a65 - a31*a44*a55*a62 - a31*a45*a52*a64 + a31*a45*a54*a62 + a32*a41*a54*a65 - a32*a41*a55*a64 - a32*a44*a51*a65 + a32*a44*a55*a61 + a32*a45*a51*a64 - a32*a45*a54*a61 - a34*a41*a52*a65 + a34*a41*a55*a62 + a34*a42*a51*a65 - a34*a42*a55*a61 - a34*a45*a51*a62 + a34*a45*a52*a61 + a35*a41*a52*a64 - a35*a41*a54*a62 - a35*a42*a51*a64 + a35*a42*a54*a61 + a35*a44*a51*a62 - a35*a44*a52*a61)*a23 + (a31*a43*a54*a65 - a31*a43*a55*a64 - a31*a44*a53*a65 + a31*a44*a55*a63 + a31*a45*a53*a64 - a31*a45*a54*a63 - a33*a41*a54*a65 + a33*a41*a55*a64 + a33*a44*a51*a65 - a33*a44*a55*a61 - a33*a45*a51*a64 + a33*a45*a54*a61 + a34*a41*a53*a65 - a34*a41*a55*a63 - a34*a43*a51*a65 + a34*a43*a55*a61 + a34*a45*a51*a63 - a34*a45*a53*a61 - a35*a41*a53*a64 + a35*a41*a54*a63 + a35*a43*a51*a64 - a35*a43*a54*a61 - a35*a44*a51*a63 + a35*a44*a53*a61)*a22 + (a32*a43*a55*a64 - a32*a43*a54*a65 + a32*a44*a53*a65 - a32*a44*a55*a63 - a32*a45*a53*a64 + a32*a45*a54*a63 + a33*a42*a54*a65 - a33*a42*a55*a64 - a33*a44*a52*a65 + a33*a44*a55*a62 + a33*a45*a52*a64 - a33*a45*a54*a62 - a34*a42*a53*a65 + a34*a42*a55*a63 + a34*a43*a52*a65 - a34*a43*a55*a62 - a34*a45*a52*a63 + a34*a45*a53*a62 + a35*a42*a53*a64 - a35*a42*a54*a63 - a35*a43*a52*a64 + a35*a43*a54*a62 + a35*a44*a52*a63 - a35*a44*a53*a62)*a21)*a16 
	+ ((a31*a42*a53*a64 - a31*a42*a54*a63 - a31*a43*a52*a64 + a31*a43*a54*a62 + a31*a44*a52*a63 - a31*a44*a53*a62 - a32*a41*a53*a64 + a32*a41*a54*a63 + a32*a43*a51*a64 - a32*a43*a54*a61 - a32*a44*a51*a63 + a32*a44*a53*a61 + a33*a41*a52*a64 - a33*a41*a54*a62 - a33*a42*a51*a64 + a33*a42*a54*a61 + a33*a44*a51*a62 - a33*a44*a52*a61 - a34*a41*a52*a63 + a34*a41*a53*a62 + a34*a42*a51*a63 - a34*a42*a53*a61 - a34*a43*a51*a62 + a34*a43*a52*a61)*a26 + (a31*a42*a56*a63 - a31*a42*a53*a66 + a31*a43*a52*a66 - a31*a43*a56*a62 - a31*a46*a52*a63 + a31*a46*a53*a62 + a32*a41*a53*a66 - a32*a41*a56*a63 - a32*a43*a51*a66 + a32*a43*a56*a61 + a32*a46*a51*a63 - a32*a46*a53*a61 - a33*a41*a52*a66 + a33*a41*a56*a62 + a33*a42*a51*a66 - a33*a42*a56*a61 - a33*a46*a51*a62 + a33*a46*a52*a61 + a36*a41*a52*a63 - a36*a41*a53*a62 - a36*a42*a51*a63 + a36*a42*a53*a61 + a36*a43*a51*a62 - a36*a43*a52*a61)*a24 + (a31*a42*a54*a66 - a31*a42*a56*a64 - a31*a44*a52*a66 + a31*a44*a56*a62 + a31*a46*a52*a64 - a31*a46*a54*a62 - a32*a41*a54*a66 + a32*a41*a56*a64 + a32*a44*a51*a66 - a32*a44*a56*a61 - a32*a46*a51*a64 + a32*a46*a54*a61 + a34*a41*a52*a66 - a34*a41*a56*a62 - a34*a42*a51*a66 + a34*a42*a56*a61 + a34*a46*a51*a62 - a34*a46*a52*a61 - a36*a41*a52*a64 + a36*a41*a54*a62 + a36*a42*a51*a64 - a36*a42*a54*a61 - a36*a44*a51*a62 + a36*a44*a52*a61)*a23 + (a31*a43*a56*a64 - a31*a43*a54*a66 + a31*a44*a53*a66 - a31*a44*a56*a63 - a31*a46*a53*a64 + a31*a46*a54*a63 + a33*a41*a54*a66 - a33*a41*a56*a64 - a33*a44*a51*a66 + a33*a44*a56*a61 + a33*a46*a51*a64 - a33*a46*a54*a61 - a34*a41*a53*a66 + a34*a41*a56*a63 + a34*a43*a51*a66 - a34*a43*a56*a61 - a34*a46*a51*a63 + a34*a46*a53*a61 + a36*a41*a53*a64 - a36*a41*a54*a63 - a36*a43*a51*a64 + a36*a43*a54*a61 + a36*a44*a51*a63 - a36*a44*a53*a61)*a22 + (a32*a43*a54*a66 - a32*a43*a56*a64 - a32*a44*a53*a66 + a32*a44*a56*a63 + a32*a46*a53*a64 - a32*a46*a54*a63 - a33*a42*a54*a66 + a33*a42*a56*a64 + a33*a44*a52*a66 - a33*a44*a56*a62 - a33*a46*a52*a64 + a33*a46*a54*a62 + a34*a42*a53*a66 - a34*a42*a56*a63 - a34*a43*a52*a66 + a34*a43*a56*a62 + a34*a46*a52*a63 - a34*a46*a53*a62 - a36*a42*a53*a64 + a36*a42*a54*a63 + a36*a43*a52*a64 - a36*a43*a54*a62 - a36*a44*a52*a63 + a36*a44*a53*a62)*a21)*a15 
	+ ((a31*a42*a55*a63 - a31*a42*a53*a65 + a31*a43*a52*a65 - a31*a43*a55*a62 - a31*a45*a52*a63 + a31*a45*a53*a62 + a32*a41*a53*a65 - a32*a41*a55*a63 - a32*a43*a51*a65 + a32*a43*a55*a61 + a32*a45*a51*a63 - a32*a45*a53*a61 - a33*a41*a52*a65 + a33*a41*a55*a62 + a33*a42*a51*a65 - a33*a42*a55*a61 - a33*a45*a51*a62 + a33*a45*a52*a61 + a35*a41*a52*a63 - a35*a41*a53*a62 - a35*a42*a51*a63 + a35*a42*a53*a61 + a35*a43*a51*a62 - a35*a43*a52*a61)*a26 + (a31*a42*a53*a66 - a31*a42*a56*a63 - a31*a43*a52*a66 + a31*a43*a56*a62 + a31*a46*a52*a63 - a31*a46*a53*a62 - a32*a41*a53*a66 + a32*a41*a56*a63 + a32*a43*a51*a66 - a32*a43*a56*a61 - a32*a46*a51*a63 + a32*a46*a53*a61 + a33*a41*a52*a66 - a33*a41*a56*a62 - a33*a42*a51*a66 + a33*a42*a56*a61 + a33*a46*a51*a62 - a33*a46*a52*a61 - a36*a41*a52*a63 + a36*a41*a53*a62 + a36*a42*a51*a63 - a36*a42*a53*a61 - a36*a43*a51*a62 + a36*a43*a52*a61)*a25 + (a31*a42*a56*a65 - a31*a42*a55*a66 + a31*a45*a52*a66 - a31*a45*a56*a62 - a31*a46*a52*a65 + a31*a46*a55*a62 + a32*a41*a55*a66 - a32*a41*a56*a65 - a32*a45*a51*a66 + a32*a45*a56*a61 + a32*a46*a51*a65 - a32*a46*a55*a61 - a35*a41*a52*a66 + a35*a41*a56*a62 + a35*a42*a51*a66 - a35*a42*a56*a61 - a35*a46*a51*a62 + a35*a46*a52*a61 + a36*a41*a52*a65 - a36*a41*a55*a62 - a36*a42*a51*a65 + a36*a42*a55*a61 + a36*a45*a51*a62 - a36*a45*a52*a61)*a23 + (a31*a43*a55*a66 - a31*a43*a56*a65 - a31*a45*a53*a66 + a31*a45*a56*a63 + a31*a46*a53*a65 - a31*a46*a55*a63 - a33*a41*a55*a66 + a33*a41*a56*a65 + a33*a45*a51*a66 - a33*a45*a56*a61 - a33*a46*a51*a65 + a33*a46*a55*a61 + a35*a41*a53*a66 - a35*a41*a56*a63 - a35*a43*a51*a66 + a35*a43*a56*a61 + a35*a46*a51*a63 - a35*a46*a53*a61 - a36*a41*a53*a65 + a36*a41*a55*a63 + a36*a43*a51*a65 - a36*a43*a55*a61 - a36*a45*a51*a63 + a36*a45*a53*a61)*a22 + (a32*a43*a56*a65 - a32*a43*a55*a66 + a32*a45*a53*a66 - a32*a45*a56*a63 - a32*a46*a53*a65 + a32*a46*a55*a63 + a33*a42*a55*a66 - a33*a42*a56*a65 - a33*a45*a52*a66 + a33*a45*a56*a62 + a33*a46*a52*a65 - a33*a46*a55*a62 - a35*a42*a53*a66 + a35*a42*a56*a63 + a35*a43*a52*a66 - a35*a43*a56*a62 - a35*a46*a52*a63 + a35*a46*a53*a62 + a36*a42*a53*a65 - a36*a42*a55*a63 - a36*a43*a52*a65 + a36*a43*a55*a62 + a36*a45*a52*a63 - a36*a45*a53*a62)*a21)*a14 
	+ ((a31*a42*a54*a65 - a31*a42*a55*a64 - a31*a44*a52*a65 + a31*a44*a55*a62 + a31*a45*a52*a64 - a31*a45*a54*a62 - a32*a41*a54*a65 + a32*a41*a55*a64 + a32*a44*a51*a65 - a32*a44*a55*a61 - a32*a45*a51*a64 + a32*a45*a54*a61 + a34*a41*a52*a65 - a34*a41*a55*a62 - a34*a42*a51*a65 + a34*a42*a55*a61 + a34*a45*a51*a62 - a34*a45*a52*a61 - a35*a41*a52*a64 + a35*a41*a54*a62 + a35*a42*a51*a64 - a35*a42*a54*a61 - a35*a44*a51*a62 + a35*a44*a52*a61)*a26 + (a31*a42*a56*a64 - a31*a42*a54*a66 + a31*a44*a52*a66 - a31*a44*a56*a62 - a31*a46*a52*a64 + a31*a46*a54*a62 + a32*a41*a54*a66 - a32*a41*a56*a64 - a32*a44*a51*a66 + a32*a44*a56*a61 + a32*a46*a51*a64 - a32*a46*a54*a61 - a34*a41*a52*a66 + a34*a41*a56*a62 + a34*a42*a51*a66 - a34*a42*a56*a61 - a34*a46*a51*a62 + a34*a46*a52*a61 + a36*a41*a52*a64 - a36*a41*a54*a62 - a36*a42*a51*a64 + a36*a42*a54*a61 + a36*a44*a51*a62 - a36*a44*a52*a61)*a25 + (a31*a42*a55*a66 - a31*a42*a56*a65 - a31*a45*a52*a66 + a31*a45*a56*a62 + a31*a46*a52*a65 - a31*a46*a55*a62 - a32*a41*a55*a66 + a32*a41*a56*a65 + a32*a45*a51*a66 - a32*a45*a56*a61 - a32*a46*a51*a65 + a32*a46*a55*a61 + a35*a41*a52*a66 - a35*a41*a56*a62 - a35*a42*a51*a66 + a35*a42*a56*a61 + a35*a46*a51*a62 - a35*a46*a52*a61 - a36*a41*a52*a65 + a36*a41*a55*a62 + a36*a42*a51*a65 - a36*a42*a55*a61 - a36*a45*a51*a62 + a36*a45*a52*a61)*a24 + (a31*a44*a56*a65 - a31*a44*a55*a66 + a31*a45*a54*a66 - a31*a45*a56*a64 - a31*a46*a54*a65 + a31*a46*a55*a64 + a34*a41*a55*a66 - a34*a41*a56*a65 - a34*a45*a51*a66 + a34*a45*a56*a61 + a34*a46*a51*a65 - a34*a46*a55*a61 - a35*a41*a54*a66 + a35*a41*a56*a64 + a35*a44*a51*a66 - a35*a44*a56*a61 - a35*a46*a51*a64 + a35*a46*a54*a61 + a36*a41*a54*a65 - a36*a41*a55*a64 - a36*a44*a51*a65 + a36*a44*a55*a61 + a36*a45*a51*a64 - a36*a45*a54*a61)*a22 + (a32*a44*a55*a66 - a32*a44*a56*a65 - a32*a45*a54*a66 + a32*a45*a56*a64 + a32*a46*a54*a65 - a32*a46*a55*a64 - a34*a42*a55*a66 + a34*a42*a56*a65 + a34*a45*a52*a66 - a34*a45*a56*a62 - a34*a46*a52*a65 + a34*a46*a55*a62 + a35*a42*a54*a66 - a35*a42*a56*a64 - a35*a44*a52*a66 + a35*a44*a56*a62 + a35*a46*a52*a64 - a35*a46*a54*a62 - a36*a42*a54*a65 + a36*a42*a55*a64 + a36*a44*a52*a65 - a36*a44*a55*a62 - a36*a45*a52*a64 + a36*a45*a54*a62)*a21)*a13 
	+ ((a31*a43*a55*a64 - a31*a43*a54*a65 + a31*a44*a53*a65 - a31*a44*a55*a63 - a31*a45*a53*a64 + a31*a45*a54*a63 + a33*a41*a54*a65 - a33*a41*a55*a64 - a33*a44*a51*a65 + a33*a44*a55*a61 + a33*a45*a51*a64 - a33*a45*a54*a61 - a34*a41*a53*a65 + a34*a41*a55*a63 + a34*a43*a51*a65 - a34*a43*a55*a61 - a34*a45*a51*a63 + a34*a45*a53*a61 + a35*a41*a53*a64 - a35*a41*a54*a63 - a35*a43*a51*a64 + a35*a43*a54*a61 + a35*a44*a51*a63 - a35*a44*a53*a61)*a26 + (a31*a43*a54*a66 - a31*a43*a56*a64 - a31*a44*a53*a66 + a31*a44*a56*a63 + a31*a46*a53*a64 - a31*a46*a54*a63 - a33*a41*a54*a66 + a33*a41*a56*a64 + a33*a44*a51*a66 - a33*a44*a56*a61 - a33*a46*a51*a64 + a33*a46*a54*a61 + a34*a41*a53*a66 - a34*a41*a56*a63 - a34*a43*a51*a66 + a34*a43*a56*a61 + a34*a46*a51*a63 - a34*a46*a53*a61 - a36*a41*a53*a64 + a36*a41*a54*a63 + a36*a43*a51*a64 - a36*a43*a54*a61 - a36*a44*a51*a63 + a36*a44*a53*a61)*a25 + (a31*a43*a56*a65 - a31*a43*a55*a66 + a31*a45*a53*a66 - a31*a45*a56*a63 - a31*a46*a53*a65 + a31*a46*a55*a63 + a33*a41*a55*a66 - a33*a41*a56*a65 - a33*a45*a51*a66 + a33*a45*a56*a61 + a33*a46*a51*a65 - a33*a46*a55*a61 - a35*a41*a53*a66 + a35*a41*a56*a63 + a35*a43*a51*a66 - a35*a43*a56*a61 - a35*a46*a51*a63 + a35*a46*a53*a61 + a36*a41*a53*a65 - a36*a41*a55*a63 - a36*a43*a51*a65 + a36*a43*a55*a61 + a36*a45*a51*a63 - a36*a45*a53*a61)*a24 + (a31*a44*a55*a66 - a31*a44*a56*a65 - a31*a45*a54*a66 + a31*a45*a56*a64 + a31*a46*a54*a65 - a31*a46*a55*a64 - a34*a41*a55*a66 + a34*a41*a56*a65 + a34*a45*a51*a66 - a34*a45*a56*a61 - a34*a46*a51*a65 + a34*a46*a55*a61 + a35*a41*a54*a66 - a35*a41*a56*a64 - a35*a44*a51*a66 + a35*a44*a56*a61 + a35*a46*a51*a64 - a35*a46*a54*a61 - a36*a41*a54*a65 + a36*a41*a55*a64 + a36*a44*a51*a65 - a36*a44*a55*a61 - a36*a45*a51*a64 + a36*a45*a54*a61)*a23 + (a33*a44*a56*a65 - a33*a44*a55*a66 + a33*a45*a54*a66 - a33*a45*a56*a64 - a33*a46*a54*a65 + a33*a46*a55*a64 + a34*a43*a55*a66 - a34*a43*a56*a65 - a34*a45*a53*a66 + a34*a45*a56*a63 + a34*a46*a53*a65 - a34*a46*a55*a63 - a35*a43*a54*a66 + a35*a43*a56*a64 + a35*a44*a53*a66 - a35*a44*a56*a63 - a35*a46*a53*a64 + a35*a46*a54*a63 + a36*a43*a54*a65 - a36*a43*a55*a64 - a36*a44*a53*a65 + a36*a44*a55*a63 + a36*a45*a53*a64 - a36*a45*a54*a63)*a21)*a12 
	+ ((a32*a43*a54*a65 - a32*a43*a55*a64 - a32*a44*a53*a65 + a32*a44*a55*a63 + a32*a45*a53*a64 - a32*a45*a54*a63 - a33*a42*a54*a65 + a33*a42*a55*a64 + a33*a44*a52*a65 - a33*a44*a55*a62 - a33*a45*a52*a64 + a33*a45*a54*a62 + a34*a42*a53*a65 - a34*a42*a55*a63 - a34*a43*a52*a65 + a34*a43*a55*a62 + a34*a45*a52*a63 - a34*a45*a53*a62 - a35*a42*a53*a64 + a35*a42*a54*a63 + a35*a43*a52*a64 - a35*a43*a54*a62 - a35*a44*a52*a63 + a35*a44*a53*a62)*a26 + (a32*a43*a56*a64 - a32*a43*a54*a66 + a32*a44*a53*a66 - a32*a44*a56*a63 - a32*a46*a53*a64 + a32*a46*a54*a63 + a33*a42*a54*a66 - a33*a42*a56*a64 - a33*a44*a52*a66 + a33*a44*a56*a62 + a33*a46*a52*a64 - a33*a46*a54*a62 - a34*a42*a53*a66 + a34*a42*a56*a63 + a34*a43*a52*a66 - a34*a43*a56*a62 - a34*a46*a52*a63 + a34*a46*a53*a62 + a36*a42*a53*a64 - a36*a42*a54*a63 - a36*a43*a52*a64 + a36*a43*a54*a62 + a36*a44*a52*a63 - a36*a44*a53*a62)*a25 + (a32*a43*a55*a66 - a32*a43*a56*a65 - a32*a45*a53*a66 + a32*a45*a56*a63 + a32*a46*a53*a65 - a32*a46*a55*a63 - a33*a42*a55*a66 + a33*a42*a56*a65 + a33*a45*a52*a66 - a33*a45*a56*a62 - a33*a46*a52*a65 + a33*a46*a55*a62 + a35*a42*a53*a66 - a35*a42*a56*a63 - a35*a43*a52*a66 + a35*a43*a56*a62 + a35*a46*a52*a63 - a35*a46*a53*a62 - a36*a42*a53*a65 + a36*a42*a55*a63 + a36*a43*a52*a65 - a36*a43*a55*a62 - a36*a45*a52*a63 + a36*a45*a53*a62)*a24 + (a32*a44*a56*a65 - a32*a44*a55*a66 + a32*a45*a54*a66 - a32*a45*a56*a64 - a32*a46*a54*a65 + a32*a46*a55*a64 + a34*a42*a55*a66 - a34*a42*a56*a65 - a34*a45*a52*a66 + a34*a45*a56*a62 + a34*a46*a52*a65 - a34*a46*a55*a62 - a35*a42*a54*a66 + a35*a42*a56*a64 + a35*a44*a52*a66 - a35*a44*a56*a62 - a35*a46*a52*a64 + a35*a46*a54*a62 + a36*a42*a54*a65 - a36*a42*a55*a64 - a36*a44*a52*a65 + a36*a44*a55*a62 + a36*a45*a52*a64 - a36*a45*a54*a62)*a23 + (a33*a44*a55*a66 - a33*a44*a56*a65 - a33*a45*a54*a66 + a33*a45*a56*a64 + a33*a46*a54*a65 - a33*a46*a55*a64 - a34*a43*a55*a66 + a34*a43*a56*a65 + a34*a45*a53*a66 - a34*a45*a56*a63 - a34*a46*a53*a65 + a34*a46*a55*a63 + a35*a43*a54*a66 - a35*a43*a56*a64 - a35*a44*a53*a66 + a35*a44*a56*a63 + a35*a46*a53*a64 - a35*a46*a54*a63 - a36*a43*a54*a65 + a36*a43*a55*a64 + a36*a44*a53*a65 - a36*a44*a55*a63 - a36*a45*a53*a64 + a36*a45*a54*a63)*a22)*a11;

END_FUNCTION

// ---- MatrixLib/invMat6.TcPOU
FUNCTION invMat6 : bool
VAR_IN_OUT CONSTANT
	mat :Mat6d;
END_VAR
VAR_IN_OUT
	invMat : Mat6d;
END_VAR
VAR
	n:INT:=6;
	m:INT:=1;
	b :ARRAY[1..6] OF LREAL := [6(0)];
	indxc,indxr, ipiv:ARRAY[1..6] OF INT := [6(0)];

	
	i,icol, irow, j,k,l,ll: INT;
	big, dum, pivinv,tmp: LREAL;
END_VAR

invMat := mat;
FOR i:=1 TO n DO   
    big:=0.0;
    FOR j:=1 TO n DO  
        IF (ipiv[j] <> 1) THEN
            FOR k:=1 TO n DO 
                IF (ipiv[k] = 0) THEN
                    IF (ABS(invMat[j,k]) >= big) THEN
                        big:=ABS(invMat[j,k]);
                        irow:=j;
                        icol:=k;
                    END_IF
                END_IF
            END_FOR
        END_IF
    END_FOR
    ipiv[icol]:=ipiv[icol]+1;
    
    IF (irow <> icol) THEN
        FOR l:=1 TO n DO 
            tmp:=invMat[irow,l];
            invMat[irow,l]:=invMat[icol,l];
            invMat[icol,l]:=tmp;
        END_FOR
 (*       FOR  l:=1 TO m DO  
            tmp:=b[irow,l];
            b[irow,l]:=b[icol,l];
            b[icol,l]:=tmp;
        END_FOR*)
    END_IF
	
    indxr[i]:=irow; 
    indxc[i]:=icol;
	
    IF invMat[icol,icol] = 0.0 THEN 
          invMat6:=FALSE;
		  RETURN;
    END_IF
	
    pivinv:=1.0/invMat[icol,icol];
    invMat[icol,icol]:=1.0;
    FOR l:=1 TO n DO  
        invMat[icol,l] := invMat[icol,l]*pivinv;
    END_FOR
 (*   FOR l:=1 TO m DO 
        b[icol,l] := b[icol,l]*pivinv;
    END_FOR*)
    FOR ll:=1 TO n DO  
        IF (ll <> icol) THEN 
            dum:=invMat[ll,icol];
            invMat[ll,icol]:=0.0;
            FOR l:=1 TO n DO  
                invMat[ll,l]:=invMat[ll,l] - invMat[icol,l]*dum;
            END_FOR
   (*         FOR l:=1 TO m DO  
                b[ll,l]:=b[ll,l] - b[icol,l]*dum;
            END_FOR*)
        END_IF
    END_FOR

END_FOR


FOR l:=n-1 TO 1 BY -1 DO 
    IF (indxr[l] <> indxc[l]) THEN
        FOR k:=1 TO n DO
            tmp:=invMat[k,indxr[l]];
            invMat[k,indxr[l]]:=invMat[k,indxc[l]];
            invMat[k,indxc[l]]:=tmp;
        END_FOR
    END_IF
END_FOR

invMat6:=TRUE;

END_FUNCTION

// ---- AgiMaths/DHTrans.TcPOU
FUNCTION DHTrans : ST_Frame
VAR_IN_OUT CONSTANT
	// DH parameters: alpha, a, d, DH[4]
	DH :Vec4d;
END_VAR
VAR
END_VAR

DHTrans.m_rot[1,1]:= COS(DH[4]);
DHTrans.m_rot[1,2]:=  -SIN(DH[4]);
DHTrans.m_rot[1,3]:= 0;
DHTrans.m_rot[2,1]:= COS(DH[1])*SIN(DH[4]);
DHTrans.m_rot[2,2]:= COS(DH[1])*COS(DH[4]);
DHTrans.m_rot[2,3]:= -SIN(DH[1]);
DHTrans.m_rot[3,1]:= SIN(DH[1])*SIN(DH[4]);
DHTrans.m_rot[3,2]:= SIN(DH[1])*COS(DH[4]);
DHTrans.m_rot[3,3]:= COS(DH[1]);

DHTrans.m_pos[1]:=DH[2];
DHTrans.m_pos[2]:=-DH[3]*SIN(DH[1]);
DHTrans.m_pos[3]:=DH[3]*COS(DH[1]);

END_FUNCTION

// ---- MatrixLib/cross.TcPOU
FUNCTION cross : Vec3d
VAR_IN_OUT CONSTANT
	a, b :Vec3d;
END_VAR
VAR
END_VAR

cross[1]:=a[2]*b[3]-a[3]*b[2];
cross[2]:=a[3]*b[1]-a[1]*b[3];
cross[3]:=a[1]*b[2]-a[2]*b[1];

END_FUNCTION

// ---- AgiMaths/sign.TcPOU
FUNCTION sign : int
VAR_INPUT
	value : LREAL;
END_VAR
VAR
END_VAR

IF value > 0 THEN 
	sign := 1;
ELSIF value <  0 THEN
	sign :=-1;
ELSE 
	sign :=0;
END_IF

END_FUNCTION

// ---- FBs_TrajectoryPlanning/linear_trajectory_with_quintic_polynomial_blends.TcPOU
FUNCTION_BLOCK linear_trajectory_with_quintic_polynomial_blends
VAR_INPUT
	t0,t1,q0,q1:lreal;
	t:lreal;	
END_VAR
VAR_OUTPUT
	pos:lreal;
	vel:lreal;
	acc:lreal;
	finished:BOOL;
END_VAR
VAR
	h,Tp,ratio,TS,TA:lreal;
	k1,t_qa,t_qb,qa,qb:lreal;
	
	Quintic_spline_curve_factor_1:Quintic_spline_curve_factor;
	Quintic_spline_curve_factor_2:Quintic_spline_curve_factor;
	a0,a1,a2,a3,a4,a5:ARRAY[1..2] OF lreal;	
END_VAR


h:=q1-q0;
Tp:=t1-t0;

ratio:=0.15;
Ts:=Tp*ratio;
Ta:=2*Ts;

k1:=h/(t1-t0-2*Ts);
t_qa:=t0+Ta;  qa:=q0+k1*(t_qa-(t0+Ts));
t_qb:=t1-Ta;  qb:=q0+k1*(t_qb-(t0+Ts));


//%计算第1段轨迹,五次多项式，始末位置的速度、加速度都为零
Quintic_spline_curve_factor_1(
	t0:= t0, 
	t1:= t_qa, 
	q0:= q0, 
	q1:= qa, 
	v0:= 0, 
	v1:= k1, 
	acc0:= 0, 
	acc1:= 0, 
	a0=> a0[1], 
	a1=> a1[1], 
	a2=> a2[1], 
	a3=> a3[1], 
	a4=> a4[1], 
	a5=> a5[1]);


//%计算第2段轨迹，直线




//%计算第3段轨迹，五次多项式，始末位置的速度、加速度都为零
Quintic_spline_curve_factor_2(
	t0:= t_qb, 
	t1:= t1, 	
	q0:= qb, 
	q1:= q1, 
	v0:= k1, 
	v1:= 0, 
	acc0:= 0, 
	acc1:= 0, 
	a0=> a0[2], 
	a1=> a1[2], 
	a2=> a2[2], 
	a3=> a3[2], 
	a4=> a4[2], 
	a5=> a5[2]);


	
	
	
IF (t<=t_qa)THEN
	t0:=t0;
	pos:=a0[1]+a1[1]*(t-t0)+a2[1]*EXPT((t-t0),2)+a3[1]*EXPT((t-t0),3)+a4[1]*EXPT((t-t0),4)+a5[1]*EXPT((t-t0),5);
	vel:=a1[1]+2*a2[1]*(t-t0)+3*a3[1]*EXPT((t-t0),2)+4*a4[1]*EXPT((t-t0),3)+5*a5[1]*EXPT((t-t0),4);
    acc:=2*a2[1]+6*a3[1]*(t-t0)+12*a4[1]*EXPT((t-t0),2)+20*a5[1]*EXPT((t-t0),3);
	
ELSIF (t<=t_qb) THEN
	t0:=t_qa;
	pos:=qa+k1*(t-t0);
	vel:=k1;
	acc:=0;
	
ELSIF (t<=t1)THEN	
	t0:=t_qb;
	pos:=a0[2]+a1[2]*(t-t0)+a2[2]*EXPT((t-t0),2)+a3[2]*EXPT((t-t0),3)+a4[2]*EXPT((t-t0),4)+a5[2]*EXPT((t-t0),5);
	vel:=a1[2]+2*a2[2]*(t-t0)+3*a3[2]*EXPT((t-t0),2)+4*a4[2]*EXPT((t-t0),3)+5*a5[2]*EXPT((t-t0),4);
	acc:=2*a2[2]+6*a3[2]*(t-t0)+12*a4[2]*EXPT((t-t0),2)+20*a5[2]*EXPT((t-t0),3);
END_IF


IF (t>t1) THEN
	finished:=TRUE;
	pos:=q1;
	vel:=0;
	acc:=0;
ELSE
	finished:=FALSE;
END_IF

END_FUNCTION_BLOCK

// ---- FBs_TrajectoryPlanning/Quintic_spline_curve_factor.TcPOU
FUNCTION_BLOCK Quintic_spline_curve_factor
VAR_INPUT
	t0,t1,q0,q1,v0,v1,acc0,acc1:lreal;
END_VAR

VAR_OUTPUT
	a0,a1,a2,a3,a4,a5:lreal;
END_VAR

VAR
	h,T:lreal;
END_VAR

h:=q1-q0;
T:=t1-t0;

a0:=q0;
a1:=v0;
a2:=acc0/2;
a3:=(20*h-(8*v1+12*v0)*T-(3*acc0-acc1)*EXPT(T,2))/(2*EXPT(T,3));
a4:=(-30*h+(14*v1+16*v0)*T+(3*acc0-2*acc1)*EXPT(T,2))/(2*EXPT(T,4));
a5:=(12*h-6*(v1+v0)*T+(acc1-acc0)*EXPT(T,2))/(2*EXPT(T,5));

END_FUNCTION_BLOCK

// ---- FBs_TrajectoryPlanning/OTG/FB_thirdOrdTrajFilter.TcPOU
// reference: trajectory planning for automatic machines and robots
FUNCTION_BLOCK FB_thirdOrdTrajFilter
VAR_INPUT
END_VAR
VAR_OUTPUT
END_VAR
VAR
	// command pos, vel and acc from last cycle
	m_cmdPos :LREAL;
	m_cmdVel :LREAL;
	m_cmdAcc :LREAL;
	m_cmdJerk:LREAL;
	
	// max velocity and acceleration
	m_maxV :LREAL;
	m_maxA :LREAL;
	m_maxJ :LREAL;
	
	// samping time
	m_Ts :LREAL;
	
	// middle variable
	ek,ek_dot,ek_ddot :LREAL;
	eDot_min, eDot_max, eDdot_min, eDdot_max:LREAL;
	delta, sigma, vp, vn, CapSig,uc:LREAL;
	
END_VAR

METHOD init : BOOL
VAR_INPUT
	i_curCmdPos : LREAL;
	i_curCmdVel :LREAL;
	i_curCmdAcc :LREAL;
	i_maxV : LREAL;
	i_maxA :LREAL;
	i_maxJ :LREAL;
	i_Ts :LREAL;
END_VAR
m_cmdPos:=i_curCmdPos;
m_cmdVel:=i_curCmdVel;
m_cmdAcc:=i_curCmdAcc;
m_maxV :=i_maxV;
m_maxA :=i_maxA;
m_maxJ :=i_maxJ;
m_Ts :=i_Ts;
END_METHOD

METHOD run : BOOL
VAR_INPUT
	i_targetPos, i_targetVel, i_targetAcc :LREAL;
END_VAR

VAR_OUTPUT
	o_cmdAcc, o_cmdVel, o_cmdPos:LREAL;
END_VAR
ek:=(m_cmdPos-i_targetPos)/m_maxJ;
ek_dot:=(m_cmdVel-i_targetVel)/m_maxJ;
ek_ddot:=(m_cmdAcc-i_targetAcc)/m_maxJ;

eDot_min:=(-m_maxV-i_targetVel)/m_maxJ;
eDot_max:=(m_maxV-i_targetVel)/m_maxJ;
eDdot_min:=(-m_maxA-i_targetAcc)/m_maxJ;
eDdot_max:=(m_maxA-i_targetAcc)/m_maxJ;

delta:=ek_dot+ek_ddot*ABS(ek_ddot)/2;
sigma:=ek+ek_dot*ek_ddot*sign(delta)-EXPT( ek_ddot,3)*(1-3*ABS(sign(delta)))/6+
	   sign(delta)*SQRT(2* EXPT((EXPT(ek_ddot,2)+2*ek_dot*sign(delta)),3))/4;
vp:=ek-eDdot_max*(ek_ddot*ek_ddot-2*ek_dot)/4-EXPT(ek_ddot*ek_ddot-2*ek_dot,2)/(8*eDdot_max)-ek_ddot*(3*ek_dot-ek_ddot*ek_ddot)/3;
vn:=ek-eDdot_min*(ek_ddot*ek_ddot+2*ek_dot)/4-EXPT(ek_ddot*ek_ddot+2*ek_dot,2)/(8*eDdot_min)+ek_ddot*(3*ek_dot+ek_ddot*ek_ddot)/3;

CapSig:=sigma;
IF ek_ddot<eDdot_max AND ek_dot<= (ek_ddot*ek_ddot/2-eDdot_max*eDdot_max) THEN
	CapSig:=vp;
ELSIF ek_ddot>eDdot_min AND ek_dot>= (-ek_ddot*ek_ddot/2+eDdot_min*eDdot_min) THEN
	CapSig:=vn;
END_IF

uc:=-m_maxJ*sign(CapSig+(1-ABS(sign(CapSig)))*(delta+(1-ABS(sign(delta)))*ek_ddot));
m_cmdJerk:=MAX(uv(eDot_min),MIN(uc,uv(eDot_max)));

o_cmdAcc:=m_cmdAcc+m_cmdJerk*m_Ts;
o_cmdVel:=m_cmdVel+(o_cmdAcc+m_cmdAcc)*m_Ts/2;
o_cmdPos:=m_cmdPos+(o_cmdVel+m_cmdVel)*m_Ts/2;
END_METHOD

METHOD PROTECTED uv : LREAL
VAR_INPUT
	in :LREAL;
END_VAR
VAR
	ua_min, ua_max, sigmaV,ucv :LREAL;
END_VAR
ua_min:=-m_maxJ*sign(ek_ddot-eDdot_min);
ua_max:=-m_maxJ*sign(ek_ddot-eDdot_max);
sigmaV:=ek_ddot*ABS(ek_ddot)+2*(ek_dot-in);
ucv:=-m_maxJ*sign(sigmaV+(1-ABS(sign(sigmaV)))*ek_ddot);
uv:=MAX(ua_min,MIN(ucv,ua_max));
END_METHOD

END_FUNCTION_BLOCK

// ---- FBs_TrajectoryPlanning/quintic_spline_curve.TcPOU
FUNCTION_BLOCK quintic_spline_curve
VAR_INPUT
	t0,t1,q0,q1:lreal;
	t:lreal;	
END_VAR
VAR_OUTPUT
	pos:lreal;
	vel:lreal;
	acc:lreal;
	finished:BOOL:=FALSE;
END_VAR
VAR
	h,Tp:lreal;
	a0,a1,a2,a3,a4,a5:lreal;
	Quintic_spline_curve_factor_1:Quintic_spline_curve_factor;
END_VAR


h:=q1-q0;
Tp:=t1-t0;

Quintic_spline_curve_factor_1(
	t0:= t0, 
	t1:= t1, 
	q0:= q0, 
	q1:= q1, 
	v0:= 0, 
	v1:= 0, 
	acc0:= 0, 
	acc1:= 0, 
	a0=> a0, 
	a1=> a1, 
	a2=> a2, 
	a3=> a3, 
	a4=> a4, 
	a5=> a5);


IF (t<=t1) THEN
	pos:=a0+a1*(t-t0)+a2*EXPT((t-t0),2)+a3*EXPT((t-t0),3)+a4*EXPT((t-t0),4)+a5*EXPT((t-t0),5);
	vel:=a1+2*a2*(t-t0)+3*a3*EXPT((t-t0),2)+4*a4*EXPT((t-t0),3)+5*a5*EXPT((t-t0),4);
	acc:=2*a2+6*a3*(t-t0)+12*a4*EXPT((t-t0),2)+20*a5*EXPT((t-t0),3);
END_IF

IF (t>t1) THEN
	finished:=TRUE;
	pos:=q1;
	vel:=0;
	acc:=0;
ELSE
	finished:=FALSE;
END_IF

END_FUNCTION_BLOCK

// ---- FBs_TrajectoryPlanning/TrapezoIDal_velocity_trajectory.TcPOU
FUNCTION_BLOCK TrapezoIDal_velocity_trajectory
VAR_INPUT
	t0,q0,q1:lreal;
	a_max,v_max:lreal;
	t:lreal;
END_VAR
VAR_OUTPUT
	pos:lreal;
	vel:lreal;
	acc:lreal;
	finished:BOOL;
END_VAR
VAR
	h,V_v,A_a:lreal;
	Tp,Ta:lreal;
	t1:lreal;
END_VAR


h:=q1-q0;

V_v:=V_max;
A_a:=A_max;
IF(h<0) THEN
    V_v:=-V_max;
    A_a:=-A_max;
END_IF


//%step1,根据给定参数，计算加速时间、总时间
IF(ABS(h)>=(V_v*V_v/ABS(A_a))) THEN
    Tp:=(h*A_a+V_v*V_v)/(A_a*V_v);
    Ta:=V_v/A_a; 
	t1:=t0+Tp;
	
	IF (t>t0) AND (t<=t0+Ta) THEN
		pos:=q0+0.5*A_a*EXPT(t-t0,2);
        vel:=A_a*(t-t0);
        acc:=A_a;	
	ELSIF (t>t0+Ta) AND (t<=t1-Ta) THEN
		pos:=q0+A_a*Ta*(t-t0-Ta/2);
        vel:=A_a*Ta;
        acc:=0;	
	ELSIF (t<=t1) THEN
		pos:=q1-0.5*A_a*EXPT(t1-t,2);
        vel:=A_a*(t1-t);
        acc:=-A_a;	
	END_IF
   
	IF (t>t1) THEN
		finished:=TRUE;
		pos:=q1;
		vel:=0;
		acc:=0;
	ELSE
		finished:=FALSE;
	END_IF
	
	
ELSE	
    //%step2,没有匀速阶段
    Ta:=SQRT(h/A_a);
    Tp:=2*Ta;
	t1:=t0+Tp;
	
	IF (t>t0) AND (t<=(t0+Ta)) THEN
		pos:=q0+0.5*A_a*EXPT((t-t0),2);
        vel:=A_a*(t-t0);
        acc:=A_a;
	ELSIF (t<=t1) THEN
		pos:=q1-0.5*A_a*EXPT(t1-t,2);
        vel:=A_a*(t1-t);
        acc:=-A_a;
	END_IF
		
	IF (t>t1) THEN
		finished:=TRUE;
		pos:=q1;
		vel:=0;
		acc:=0;
	ELSE
		finished:=FALSE;
	END_IF
		
END_IF

END_FUNCTION_BLOCK

// ---- AgiMaths/multiNumVec3.TcPOU
FUNCTION multiNumVec3 : Vec3d
VAR_IN_OUT CONSTANT
	i_num :LREAL;
	i_vec:Vec3d;
END_VAR
VAR
	i: INT ;
END_VAR

FOR i:=1 TO 3 DO 
	multiNumVec3[i]:=i_vec[i]*i_num;
END_FOR

END_FUNCTION

// ---- AgiMaths/normVec3.TcPOU
FUNCTION normVec3 : LREAL
VAR_IN_OUT CONSTANT
	vec3 :Vec3d;
END_VAR
VAR
END_VAR

normVec3:=SQRT(vec3[1]*vec3[1]+vec3[2]*vec3[2]+vec3[3]*vec3[3]);

END_FUNCTION

// ---- MatrixLib/Det5.TcPOU
FUNCTION Det5 : LREAL
VAR_IN_OUT CONSTANT
	mat: Mat5d;
END_VAR
VAR
	a11,a12,a13,a14,a15,a16:LREAL;
	a21,a22,a23,a24,a25,a26:LREAL;
	a31,a32,a33,a34,a35,a36:LREAL;
	a41,a42,a43,a44,a45,a46:LREAL;
	a51,a52,a53,a54,a55,a56:LREAL;
	a61,a62,a63,a64,a65,a66:LREAL;
END_VAR



//***************求取5X5矩阵的秩****************//
a11:=mat[1,1];
a12:=mat[1,2];
a13:=mat[1,3];
a14:=mat[1,4];
a15:=mat[1,5];

a21:=mat[2,1];
a22:=mat[2,2];
a23:=mat[2,3];
a24:=mat[2,4];
a25:=mat[2,5];

a31:=mat[3,1];
a32:=mat[3,2];
a33:=mat[3,3];
a34:=mat[3,4];
a35:=mat[3,5];

a41:=mat[4,1];
a42:=mat[4,2];
a43:=mat[4,3];
a44:=mat[4,4];
a45:=mat[4,5];

a51:=mat[5,1];
a52:=mat[5,2];
a53:=mat[5,3];
a54:=mat[5,4];
a55:=mat[5,5];

//Det5:=a11*a22*a33*a44*a55 - a11*a22*a33*a45*a54 - a11*a22*a34*a43*a55 + a11*a22*a34*a45*a53 + a11*a22*a35*a43*a54 - a11*a22*a35*a44*a53 - a11*a23*a32*a44*a55 + a11*a23*a32*a45*a54 + a11*a23*a34*a42*a55 - a11*a23*a34*a45*a52 - a11*a23*a35*a42*a54 + a11*a23*a35*a44*a52 + a11*a24*a32*a43*a55 - a11*a24*a32*a45*a53 - a11*a24*a33*a42*a55 + a11*a24*a33*a45*a52 + a11*a24*a35*a42*a53 - a11*a24*a35*a43*a52 - a11*a25*a32*a43*a54 + a11*a25*a32*a44*a53 + a11*a25*a33*a42*a54 - a11*a25*a33*a44*a52 - a11*a25*a34*a42*a53 + a11*a25*a34*a43*a52 - a12*a21*a33*a44*a55 + a12*a21*a33*a45*a54 + a12*a21*a34*a43*a55 - a12*a21*a34*a45*a53 - a12*a21*a35*a43*a54 + a12*a21*a35*a44*a53 + a12*a23*a31*a44*a55 - a12*a23*a31*a45*a54 - a12*a23*a34*a41*a55 + a12*a23*a34*a45*a51 + a12*a23*a35*a41*a54 - a12*a23*a35*a44*a51 - a12*a24*a31*a43*a55 + a12*a24*a31*a45*a53 + a12*a24*a33*a41*a55 - a12*a24*a33*a45*a51 - a12*a24*a35*a41*a53 + a12*a24*a35*a43*a51 + a12*a25*a31*a43*a54 - a12*a25*a31*a44*a53 - a12*a25*a33*a41*a54 + a12*a25*a33*a44*a51 + a12*a25*a34*a41*a53 - a12*a25*a34*a43*a51 + a13*a21*a32*a44*a55 - a13*a21*a32*a45*a54 - a13*a21*a34*a42*a55 + a13*a21*a34*a45*a52 + a13*a21*a35*a42*a54 - a13*a21*a35*a44*a52 - a13*a22*a31*a44*a55 + a13*a22*a31*a45*a54 + a13*a22*a34*a41*a55 - a13*a22*a34*a45*a51 - a13*a22*a35*a41*a54 + a13*a22*a35*a44*a51 + a13*a24*a31*a42*a55 - a13*a24*a31*a45*a52 - a13*a24*a32*a41*a55 + a13*a24*a32*a45*a51 + a13*a24*a35*a41*a52 - a13*a24*a35*a42*a51 - a13*a25*a31*a42*a54 + a13*a25*a31*a44*a52 + a13*a25*a32*a41*a54 - a13*a25*a32*a44*a51 - a13*a25*a34*a41*a52 + a13*a25*a34*a42*a51 - a14*a21*a32*a43*a55 + a14*a21*a32*a45*a53 + a14*a21*a33*a42*a55 - a14*a21*a33*a45*a52 - a14*a21*a35*a42*a53 + a14*a21*a35*a43*a52 + a14*a22*a31*a43*a55 - a14*a22*a31*a45*a53 - a14*a22*a33*a41*a55 + a14*a22*a33*a45*a51 + a14*a22*a35*a41*a53 - a14*a22*a35*a43*a51 - a14*a23*a31*a42*a55 + a14*a23*a31*a45*a52 + a14*a23*a32*a41*a55 - a14*a23*a32*a45*a51 - a14*a23*a35*a41*a52 + a14*a23*a35*a42*a51 + a14*a25*a31*a42*a53 - a14*a25*a31*a43*a52 - a14*a25*a32*a41*a53 + a14*a25*a32*a43*a51 + a14*a25*a33*a41*a52 - a14*a25*a33*a42*a51 + a15*a21*a32*a43*a54 - a15*a21*a32*a44*a53 - a15*a21*a33*a42*a54 + a15*a21*a33*a44*a52 + a15*a21*a34*a42*a53 - a15*a21*a34*a43*a52 - a15*a22*a31*a43*a54 + a15*a22*a31*a44*a53 + a15*a22*a33*a41*a54 - a15*a22*a33*a44*a51 - a15*a22*a34*a41*a53 + a15*a22*a34*a43*a51 + a15*a23*a31*a42*a54 - a15*a23*a31*a44*a52 - a15*a23*a32*a41*a54 + a15*a23*a32*a44*a51 + a15*a23*a34*a41*a52 - a15*a23*a34*a42*a51 - a15*a24*a31*a42*a53 + a15*a24*a31*a43*a52 + a15*a24*a32*a41*a53 - a15*a24*a32*a43*a51 - a15*a24*a33*a41*a52 + a15*a24*a33*a42*a51;
Det5:=((a31*a43*a52 - a31*a42*a53 + a32*a41*a53 - a32*a43*a51 - a33*a41*a52 + a33*a42*a51)*a24 + (a31*a42*a54 - a31*a44*a52 - a32*a41*a54 + a32*a44*a51 + a34*a41*a52 - a34*a42*a51)*a23 + (a31*a44*a53 - a31*a43*a54 + a33*a41*a54 - a33*a44*a51 - a34*a41*a53 + a34*a43*a51)*a22 + (a32*a43*a54 - a32*a44*a53 - a33*a42*a54 + a33*a44*a52 + a34*a42*a53 - a34*a43*a52)*a21)*a15 
	+ ((a31*a42*a53 - a31*a43*a52 - a32*a41*a53 + a32*a43*a51 + a33*a41*a52 - a33*a42*a51)*a25 + (a31*a45*a52 - a31*a42*a55 + a32*a41*a55 - a32*a45*a51 - a35*a41*a52 + a35*a42*a51)*a23 + (a31*a43*a55 - a31*a45*a53 - a33*a41*a55 + a33*a45*a51 + a35*a41*a53 - a35*a43*a51)*a22 + (a32*a45*a53 - a32*a43*a55 + a33*a42*a55 - a33*a45*a52 - a35*a42*a53 + a35*a43*a52)*a21)*a14 
	+ ((a31*a44*a52 - a31*a42*a54 + a32*a41*a54 - a32*a44*a51 - a34*a41*a52 + a34*a42*a51)*a25 + (a31*a42*a55 - a31*a45*a52 - a32*a41*a55 + a32*a45*a51 + a35*a41*a52 - a35*a42*a51)*a24 + (a31*a45*a54 - a31*a44*a55 + a34*a41*a55 - a34*a45*a51 - a35*a41*a54 + a35*a44*a51)*a22 + (a32*a44*a55 - a32*a45*a54 - a34*a42*a55 + a34*a45*a52 + a35*a42*a54 - a35*a44*a52)*a21)*a13 
	+ ((a31*a43*a54 - a31*a44*a53 - a33*a41*a54 + a33*a44*a51 + a34*a41*a53 - a34*a43*a51)*a25 + (a31*a45*a53 - a31*a43*a55 + a33*a41*a55 - a33*a45*a51 - a35*a41*a53 + a35*a43*a51)*a24 + (a31*a44*a55 - a31*a45*a54 - a34*a41*a55 + a34*a45*a51 + a35*a41*a54 - a35*a44*a51)*a23 + (a33*a45*a54 - a33*a44*a55 + a34*a43*a55 - a34*a45*a53 - a35*a43*a54 + a35*a44*a53)*a21)*a12 
	+ ((a32*a44*a53 - a32*a43*a54 + a33*a42*a54 - a33*a44*a52 - a34*a42*a53 + a34*a43*a52)*a25 + (a32*a43*a55 - a32*a45*a53 - a33*a42*a55 + a33*a45*a52 + a35*a42*a53 - a35*a43*a52)*a24 + (a32*a45*a54 - a32*a44*a55 + a34*a42*a55 - a34*a45*a52 - a35*a42*a54 + a35*a44*a52)*a23 + (a33*a44*a55 - a33*a45*a54 - a34*a43*a55 + a34*a45*a53 + a35*a43*a54 - a35*a44*a53)*a22)*a11;

END_FUNCTION

// ---- MatrixLib/invMat6Old.TcPOU
FUNCTION invMat6Old : bool
VAR_IN_OUT CONSTANT
	mat :Mat6d;
END_VAR

VAR_IN_OUT
	invMat :Mat6d;
END_VAR
VAR
	dim : INT :=6;
	i,j,k,h:INT;
	m,n :INT;
	cofactorMat : Mat5d;
	adjointMat :Mat6d;
	matDet :LREAL;
END_VAR

matDet :=Det6(mat);
IF matDet=0 THEN
	invMat6Old:=FALSE;
	RETURN;
END_IF

FOR i :=1 TO dim DO
	FOR j:=1 TO dim DO
		// get cofactor mat
		m:=1;
		n:=1;
		FOR k:=1 TO dim DO
			FOR h:=1 TO dim DO
				IF k<>i AND h <> j THEN
					cofactorMat[m,n]:=mat[k,h];
					n:=n+1;
					IF n>=dim THEN
						m:=m+1;
						n:=1;
					END_IF
				END_IF
			END_FOR
		END_FOR
		
		adjointMat[i,j]:=EXPT(-1,i+j)*Det5(cofactorMat);
	END_FOR
END_FOR

FOR i :=1 TO dim DO
	FOR j:=1 TO dim DO
		invMat[i,j]:=adjointMat[j,i]/matDet;
	END_FOR
END_FOR

invMat6Old:=TRUE;

END_FUNCTION

// ---- MatrixLib/Mat3T.TcPOU
FUNCTION Mat3T : Mat3d
VAR_IN_OUT CONSTANT
	mat :Mat3d;
END_VAR
VAR
END_VAR

Mat3T[1,1]:=mat[1,1];
Mat3T[1,2]:=mat[2,1];
Mat3T[1,3]:=mat[3,1];
Mat3T[2,1]:=mat[1,2];
Mat3T[2,2]:=mat[2,2];
Mat3T[2,3]:=mat[3,2];
Mat3T[3,1]:=mat[1,3];
Mat3T[3,2]:=mat[2,3];
Mat3T[3,3]:=mat[3,3];

END_FUNCTION

// ---- MatrixLib/matSelfSub.TcPOU
// A -=B
FUNCTION matSelfSub : BOOL
VAR_IN_OUT;
	matA :ARRAY[*,*] OF LREAL;
END_VAR

VAR_IN_OUT CONSTANT
	matB :ARRAY[*,*] OF LREAL;
END_VAR

VAR
	m,n :DINT;
	i,j, k :DINT;
 
END_VAR

m:=UPPER_BOUND(matA,1);
n:= UPPER_BOUND(matA,2);
FOR i:=1 TO m DO
	FOR j:=1 TO n DO
		matA[i,j]:=matA[i,j]-matB[i,j];
	END_FOR
END_FOR

END_FUNCTION

// ---- MatrixLib/matAdd.TcPOU
// C = A + B;
FUNCTION matAdd : BOOL
VAR_IN_OUT;
	matA :ARRAY[*,*] OF LREAL;
END_VAR

VAR_IN_OUT CONSTANT
		matB :ARRAY[*,*] OF LREAL;
END_VAR

VAR
	m,n :DINT;
	i,j, k :DINT;
 
END_VAR

m:=UPPER_BOUND(matA,1);
n:= UPPER_BOUND(matA,2);
FOR i:=1 TO m DO
	FOR j:=1 TO n DO
		matA[i,j]:=matA[i,j]+matB[i,j];
	END_FOR
END_FOR

END_FUNCTION
